(* CODESYS project CtaAppReport_2.0.0.0.library
   Description: Report Library der CTA
   Version: 2.0.0.0
   Title: CtaAppReport
   Author: SIS
   Company: CTA
   Placeholder: CtaAppReport
   DocFormat: reStructuredText
   DefaultNamespace: CtaAppReport
   CompiledLibraryCompatibilityVersion: CODESYS V3.5 SP16 Patch 3
   LanguageModelAttribute: qualified-access-only

Project tree, tasks and I/O mapping:
  libraries: Standard, 3.5.18.0 (System); CtaAppBmk, 2.0.0.0 (CTA); CtaSysConfig, 1.0.0.2 (CTA); CtaVisSymbols, 1.0.0.0 (CTA); CtaSysEvent, 1.0.0.0 (CTA); VisuDialogs, 3.5.16.20 (System); SysFile, 3.5.17.0 (System); SysDir, 3.5.17.0 (System); VisuSymbols, 4.5.0.0 (System); StringUtils, 3.5.18.0 (System); SysTypes2 Interfaces, * (System); TextListUtils, * (System); CtaAppInfluxLog, 1.0.0.1 (CTA); CtaAppTime, 1.0.0.1 (CTA)
  40 Visualizations/
    visualisation REPORT_ID
    TABLE/
      visualisation VIS_REPORT_TABLE
      visualisation VIS_REPORT_TABLE_BASE
      DELETE/
        visualisation VIS_REPORT_DELETE
    PUSHLINE/
      visualisation VIS_REPORT_PUSH_LINE
      visualisation VIS_REPORT_PUSH_LINE_BASE
      visualisation VIS_REPORT_PUSH_LINE_QUERRY
    TABLE LINE/
      visualisation VIS_REPORT_TABLE_LINE_BASE
      visualisation VIS_REPORT_TABLE_LINE_QUERRY
      visualisation VIS_REPORT_TABLE_LINE
    REPORTMANAGER/
      visualisation VIS_REPORTMANAGER
      visualisation VIS_REPORTMANAGER_BASE
    HAND/
      visualisation VIS_REPORT_HAND
    ANZAHL REPORTS/
      visualisation VIS_ANZ_REPORTS_OVERALL
      Modul/
        visualisation VIS_ANZ_REPORTS_MODUL
        visualisation VIS_ANZ_REPORTS_MODUL_BASE
        visualisation VIS_ANZ_REPORTS_MODUL_QUERRY
  30 Program Organization Units/
    CSV/
      function block fbCsvHandler [ST]: metWriteDtFrom, metOpenFile, metCloseFile, FB_INIT, metFillSpace, FB_EXIT, metWriteDtTo, actInitPath, metReadCsv, proGetCountsOfReports, proGetCountOfReportsOnInit, metCreateHeader, proExportIdStart, metExportId, metResetCycleCount, proExport, proIsRegistred, metStartDone, metPrepeareStop, proDenyStop, metCyclicCall, metWriteOnChange, metDeleteHistory, metAddObjForeWriteDtFrom, metAddObjForeWriteDtTo, metAddObjForeWriteOnChange
    OBJ/
      function block fbReportObjectFactory [ST]: metQuittAllReports, metDestroyCsvReportObject, metQuittSelectedReports, metCsvGetItf, metDestroyReportObject, metGetItf, metCreateReportObject, proGetNextPos, proGetAktiveReport, proGetActiveErrorMbString, proIsThereAnAktiveError, proGetActiveWarningMbString, metReSaveAfterDelete, metGarbageControll
      function block fbReportObject [ST]: proGetReporterText, proGetReportText, proAdditionalText, proCountRetry, proIsQuitt, proIsSelected, proMaxRetry, proReportAcknowledgType, proReportId, proReportTextId, proReportTextList, proReportType, proReporterObjectId, proStateActive, proWritePosInCsv, proQuitt, metSendDataToInflux, metReportObject, proReportIn, proDtFrom, proDtTo, proSetMetaData, metDestroy, proPrio, metWriteDtFromToCsv, metWriteDtToToCsv, metSaveOnChange, metGarbage
      function fcWordToHexString [ST]
      function fcReportIdToString8 [ST]
    REPORTER/
      function block fbReportManager [ST]: proWarningText, metSyncReporter, proInfoText, proErrorText, proGetErrorNr, actInit, proGetWarningNr, proGetInfoNr, proAnzError, proAnzWarning, proAnzInfo, proTotalReports
      function block fbReporter [ST]: metGetQuitt, proAktivReport, proHandLokal, proNewReport, metReport, proGetCounts, proDoneReport, proPrio, proOptionalText
    VIS/
      function block fbReportVisu [ST]: metGetReport, metGetShowReport, actConfigFile, proQuittExtern, proMaxOffset, proOffset, actEWI, FB_INIT, metReload, actHistory, actPending, proFilterError, proFilterWarning, proFilterInfo, actCheckFilterAndSort, proAnzReportsInTable, proIdMissmatch
    function fcBmkToId [ST]
    SORT/
      function block fbSort [ST]: metSortPrio, metFilterCustom, proAnzAktiveError, proAnzAktiveInfo, proAnzAktiveReports, proAnzAktiveWarning, proAnzReportsInTable
    program REPORT [ST]
  00000000-0000-0000-0000-000000000000|D:\CoDeSys\LibrariesV3\trunk\Intern\CAA\CAA Template\3.4.0.0 draft\Placeholder.xml
  00000000-0000-0000-0000-000000000000|D:\CoDeSys\LibrariesV3\trunk\Intern\CAA\CAA Template\3.2.0.3 draft\Prefix.pdf
  00000000-0000-0000-0000-000000000000|D:\CoDeSys\LibrariesV3\trunk\Intern\CAA\CAA Template\3.5.2.0 draft\Placeholder.xml
  20 Structs/
    data type enReportType
    data type scPara
    data type scReportMetaData
    data type scReportNr
    data type stReportTextList
    data type enReportacknowledgeType
    data type enTableType
  50 Images/
  10 Documenation/
    global variables VersionHistory
    global variables readMe
  21 Interface/
    interface ITF_REPORTMANAGER: proErrorText, proGetWarningNr, metSyncReporter, proGetErrorNr, proGetInfoNr, proInfoText, proWarningText, proTotalReports
    interface ITF_REPORTOBJECT: proGetReportText, proStateActive, proIsQuitt, proIsSelected, proReportId, proMaxRetry, proCountRetry, proReportTextList, proReportTextId, proReporterObjectId, proAdditionalText, proReportType, proReportAcknowledgType, proWritePosInCsv, proGetReporterText, proReportIn, proDtTo, proDtFrom, metReportObject, proQuitt, proSetMetaData, proPrio, metDestroy, metWriteDtFromToCsv, metSaveOnChange
  11 Library Parameter/
    global variables Parameter
  12 Konstanten/
    global variables GlobalKonstant
  60 Textlisten/
    text list txtLibAp99_1Error
    text list txtLibAp99_2enTypeOfAck
    text list txtLibAp99_2Warnung
    text list txtLibAp99_3Info
    text list GlobalTextList
    text list txtNoTextList
  13 Globale Variablen/
    global variables GVL_Report
    global variables GVL_REPORT_PERSISTENT
*)

// 20 Structs/enReportType
TYPE enReportType :
(
	Info    := 0,
    Warning := 1,
    Error   := 2
);
END_TYPE

// 20 Structs/scPara
TYPE scPara :
    STRUCT
        fbxEnSafetyFernQuitt            :   CtaSysConfig.fbBOOL;
        fbuiMaxFernQuitt                :   CtaSysConfig.fbUINT;         
    END_STRUCT
END_TYPE

// 20 Structs/scReportMetaData
TYPE scReportMetaData :
    STRUCT
        xReportIn                   :   BOOL;                           // Report Input
        xActive                     :   BOOL;                           // State of Report
        xIsQuitt                    :   BOOL;                           // State of Acknowledge
        xQuitt                      :   BOOL;                           // Acknowledge Flag
        xIsSelected                 :   BOOL;                           // State of Selected in Table
        dtFrom                      :   DT;                             // Date and Time of Report happen
        dtTo                        :   DT;                             // Date and Time of Report gone
        iMaxRetry                   :   INT;                            // Max allowed Retries till Acknowledge is required
        iCountRetry                 :   INT;                            // Retries till now
        stReportTxtId               :   STRING[3];                      // Report Id fore Texlist
        stReportTextList            :   STRING[100];                    // Report TextList 
        uliReportId                 :   ULINT;                          // Report Id build out of BMK and Report Text Id. Ex: Bmk 56M111 & Id 3 = 567711103  
        enReportType                :   enReportType;                   // Type of Report
        enReportacknowledgeType     :   enReportacknowledgeType;        // Type of Report Acknowledge
        stReporterObjId             :   STRING[20];                     // Object Id of Reporter      
        stAdditionalText            :   STRING[20];                     // Additional Text
        dwWritePosInCsv             :   DWORD;                          // Position in Csv File fore write dtTo 
        usiPrio                     :   USINT;                          // Prio
    END_STRUCT
END_TYPE

// 20 Structs/scReportNr
TYPE scReportNr :
    STRUCT
        iError              :   INT;            // Error Status
        usiErrorPrio        :   USINT;
        iWarning            :   INT;            // Warning Status
        usiWarnungPrio      :   USINT;
        iInfo               :   INT;            // Info Status
        usiInfoPrio         :   USINT;
    END_STRUCT
END_TYPE

// 20 Structs/stReportTextList
TYPE stReportTextList : STRING[100]; END_TYPE

// 20 Structs/enReportacknowledgeType
TYPE enReportacknowledgeType :
(
	Auto        := 0,
    Quit        := 1,
    RetryN      := 2
);
END_TYPE

// 20 Structs/enTableType
{attribute 'qualified_only'}
{attribute 'strict'}
TYPE enTableType :
(
	PENDING_REPORTS := 0,
    HISTORY_REPORTS := 1
);
END_TYPE

// 10 Documenation/VersionHistory
(* 

.. image:: ../../Images/CTA_Logo.jpg
   :align: right
   :width: 15% 

**Vorlage**   


============ =========== =========== ============================================
**Date**     **Version** **Author**  **Change**
------------ ----------- ----------- --------------------------------------------
04.03.2021   0.0.0.0     SIS         Vorlage erstellt

============ =========== =========== ============================================


*)
VAR_GLOBAL
    stInfo : STRING:= '0.0.0.0, Vorlage, CTA';
END_VAR

// 10 Documenation/readMe
(*

**ReadMe**
 
|	**Empfehlung**
|
|	Die LibAp99aErrorManagement wird benötigt damit aus dem BMK der CTA-E-Schema eine Störungsnummer generiert werden kann. 
|	Es wird für die Ausgabe ein DINT verwendet. Die aufschlüsselung von Buchstaben wird durch die ASCI Nr ersetzt.     
|  
| *Beispiel* 
|
| BMK             =   **56M11**    
| Fehler Nr       =   01-10
| ErrorNr-Modbus  =   BMK    + Fehler Nr
| 56771101        =   567711 + 01
| 56771102        =   567711 + 02
| 56771103        =   567711 + 03
| 56771104        =   567711 + 04
| 56771105        =   567711 + 05
| 56771106        =   567711 + 06
| 56771107        =   567711 + 07 
| 56771108        =   567711 + 08
| 56771109        =   567711 + 09
| 56771110        =   567711 + 10 
|
| Wenn der Fehler keiner BMK zugeordnet werden kann, sollte von der Nr. 1000 hochgezähl werden. 
| Tiefere Nr. werden von den Bibliotheken benötigt. 
*)

VAR_GLOBAL
    xReadMeDone              :   BOOL;
END_VAR

// 13 Globale Variablen/GVL_Report
{attribute 'qualified_only'}
VAR_GLOBAL
    fbReportObjectFactory     :   fbReportObjectFactory;
    fbSort                    :   fbSort;
    fbReportVisu              :   fbReportVisu;
    (* Reports *)             
    ayReportObject            :   ARRAY[1..Parameter.diMaxObject] OF fbReportObject;
    ayItfAktiveReports        :   ARRAY[1..Parameter.diMaxObject] OF ITF_REPORTOBJECT;
    ayItfSortetReportsPrio    :   ARRAY[1..Parameter.diMaxObject] OF ITF_REPORTOBJECT;
    ayItfSortetReportsCustom  :   ARRAY[1..Parameter.diMaxObject] OF ITF_REPORTOBJECT;
    ayCsvReportObject         :   ARRAY[0..GlobalKonstant.iUpperSizeTable] OF fbReportObject;
    fbCsvHandler              :   fbCsvHandler;
    diCountHand               :   DINT;
END_VAR

// 11 Library Parameter/Parameter
{attribute 'qualified_only'}
VAR_GLOBAL CONSTANT
    diMaxObject                  :   DINT :=  50;    // Max 200
    diMaxExportsPerCycle         :   DINT :=  50;    // Kann sich auf die Zykluszeit auswirken wenn zu viele Id pro Zyklus exportiert werden
END_VAR

// 12 Konstanten/GlobalKonstant
{attribute 'qualified_only'}
VAR_GLOBAL CONSTANT
    stTextListWarning           :   stReportTextList    := 'CtaAppReport.txtLibAp99_2Warnung';
    stTextListInfo              :   stReportTextList    := 'CtaAppReport.txtLibAp99_3Info';
    iUpperSizeTable             :   INT                 := 13;   
END_VAR

// 13 Globale Variablen/GVL_REPORT_PERSISTENT
{attribute 'qualified_only'}
VAR_GLOBAL RETAIN 
	scLastErrorReport         :   scReportMetaData;
	scLastWarningReport       :   scReportMetaData;
	scLastInfoReport          :   scReportMetaData;  
END_VAR

// 21 Interface/ITF_REPORTMANAGER
INTERFACE ITF_REPORTMANAGER EXTENDS __SYSTEM.IQueryInterface

PROPERTY proErrorText : STRING[100]
GET
END_GET
END_PROPERTY

PROPERTY proGetWarningNr : INT
GET
END_GET
END_PROPERTY

METHOD metSyncReporter : BOOL
VAR_INPUT
	refFbReporter	:	REFERENCE TO fbReporter;
END_VAR
END_METHOD

PROPERTY proGetErrorNr : INT
GET
END_GET
END_PROPERTY

PROPERTY proGetInfoNr : INT
GET
END_GET
END_PROPERTY

PROPERTY proInfoText : STRING[100]
GET
END_GET
END_PROPERTY

PROPERTY proWarningText : STRING[100]
GET
END_GET
END_PROPERTY

PROPERTY proTotalReports : INT
GET
END_GET
END_PROPERTY

END_INTERFACE

// 30 Program Organization Units/REPORTER/fbReporter
FUNCTION_BLOCK FINAL fbReporter 
VAR
	diArrayReportAdr     :	DINT;
	iCountReports		 :	INT;
	tonDelay			 :	TON;
	tonReset			 :	TON;
	_stReportTextList    :	POINTER TO stReportTextList;
	_iReportID			 :  INT;
	xNewReport			 :  BOOL;
	xAktiveReport		 :  BOOL;
    xDoneReport          :  BOOL;
	_enReportType        :  enReportType;
    xHand                :  BOOL;
    usiPrio              :  USINT;
    xExportDone          :  BOOL; 
    xInitDone            :  BOOL;
END_VAR

METHOD metGetQuitt : BOOL
VAR
    ITF_REPORTOBJECT : ITF_REPORTOBJECT;
END_VAR
IF diArrayReportAdr >= 1 THEN
    IF __QUERYINTERFACE(GVL_Report.fbReportObjectFactory.metGetItf(diArrayReportAdr),ITF_REPORTOBJECT) THEN
        metGetQuitt := ITF_REPORTOBJECT.proIsQuitt;
    END_IF;
ELSE
    metGetQuitt := FALSE;
END_IF
END_METHOD

PROPERTY proAktivReport : BOOL
GET
proAktivReport := xAktiveReport;
END_GET
END_PROPERTY

PROPERTY proHandLokal : BOOL
SET
IF proHandLokal AND  NOT xHand THEN
    GVL_Report.diCountHand := GVL_Report.diCountHand + 1;
    xHand := TRUE;
ELSIF NOT proHandLokal AND xHand THEN
    GVL_Report.diCountHand := GVL_Report.diCountHand - 1;
    IF GVL_Report.diCountHand < 0 THEN
        GVL_Report.diCountHand := 0;
	END_IF;
    xHand := FALSE;    
END_IF;
END_SET
END_PROPERTY

PROPERTY INTERNAL proNewReport : BOOL
SET
xNewReport := proNewReport;
END_SET
GET
proNewReport := xNewReport;
END_GET
END_PROPERTY

METHOD FINAL metReport : BOOL
VAR_INPUT
    xSetReportIn          		:   BOOL;
    iReportID           		:   INT;
    enReportTypeIn      		:   enReportType;
    enReportAcknowledgeTypeIn   :   enReportAcknowledgeType;
	tDelay              		:   TIME;  
	ITF_BMK_IN					:	CtaAppBmk.ITF_BMK;
	pstReportTextListIn 		:	POINTER TO stReportTextList;	 
	stOptionalReportText		:	STRING[20];	
    iRetryTilReportLock 		:   INT;                            
    xResetCount         		:   BOOL;                            
	tReset						:	TIME;                 
END_VAR
VAR
    ITF_REPORTOBJECT            :   ITF_REPORTOBJECT;
END_VAR
IF xInitDone AND_THEN pstReportTextListIn <> 0 AND_THEN ITF_BMK_IN <> 0 THEN
    // Counter mit xResetCount rücksetzen wenn Count < iMaxRetry
    IF tReset > T#0MS AND_THEN enReportAcknowledgeTypeIn = enReportacknowledgeType.RetryN AND_THEN NOT xSetReportIn THEN
        tonReset.IN := iCountReports < iRetryTilReportLock AND iCountReports > 0;
        tonReset.PT	:= tReset;
        tonReset();
	ELSE
		tonReset(IN := FALSE,
				 PT := T#0MS);
    END_IF;
    IF (xResetCount OR tonReset.Q) AND_THEN iCountReports < iRetryTilReportLock AND NOT xSetReportIn  THEN
        diArrayReportAdr := 0;   
        iCountReports := 0;
        tonReset.IN := FALSE;
        tonReset.PT	:= T#0S;	 
        tonReset();
    END_IF;        
	IF xSetReportIn THEN	
		_stReportTextList    := pstReportTextListIn;	
		_iReportID 			 := iReportID;
		_enReportType		 := enReportTypeIn;
	END_IF;
	
	tonDelay.IN          := xSetReportIn;
	tonDelay.PT          := tDelay;
	tonDelay();
	(* Wenn Report nicht registriert Registrierprozess starten *)
    IF diArrayReportAdr = 0 THEN
        // Wenn tonDelay.Q aktiv Registrieren      
        IF tonDelay.Q THEN
            (* Create Report Object *)
            diArrayReportAdr := GVL_Report.fbReportObjectFactory.metCreateReportObject();   
            IF diArrayReportAdr <> 0 THEN 
                IF __QUERYINTERFACE(GVL_Report.fbReportObjectFactory.metGetItf(diArrayReportAdr),ITF_REPORTOBJECT) THEN               
                    (* Set Infos *)  
                    xNewReport := TRUE;
                    xAktiveReport := TRUE;
                    iCountReports := iCountReports + 1;
                    ITF_REPORTOBJECT.proReportType              :=  enReportTypeIn;                         // Report Type
                    ITF_REPORTOBJECT.proReportAcknowledgType    :=  enReportAcknowledgeTypeIn;              // Report Acknowledge Type
                    ITF_REPORTOBJECT.proReportTextId            :=  TO_STRING(iReportID);                   // Report Id
                    ITF_REPORTOBJECT.proReportTextList          :=  pstReportTextListIn^;                   // Report Text list
                    ITF_REPORTOBJECT.proReporterObjectId        :=  ITF_BMK_IN.proGetObjectId;              // Reporter Object Id
                    ITF_REPORTOBJECT.proSetInstancePath         :=  ITF_BMK_IN.proGetInstancePath;          // Reporter Instance Path
                    ITF_REPORTOBJECT.proMaxRetry                :=  iRetryTilReportLock;                    // Max Retries
                    ITF_REPORTOBJECT.proCountRetry              :=  iCountReports;                          // Countet Retries
                    ITF_REPORTOBJECT.proAdditionalText          :=  stOptionalReportText;                   // Additional Text
                    ITF_REPORTOBJECT.proReportIn                :=  xSetReportIn;                           // Report Input
                    ITF_REPORTOBJECT.proPrio                    :=  usiPrio;
                    ITF_REPORTOBJECT.metReportObject();                                                     // Call Object              
                END_IF                                                                 
            END_IF;
        END_IF;
    ELSE
        // Zyklische aktualisierung der Daten nach Registrierung       
        IF __QUERYINTERFACE(GVL_Report.fbReportObjectFactory.metGetItf(diArrayReportAdr),ITF_REPORTOBJECT) THEN
            IF ITF_REPORTOBJECT.proReportIn <> xSetReportIn THEN
                ITF_REPORTOBJECT.proReportIn :=  xSetReportIn;                                   // Report Input
            END_IF;
			// Nach Manuellem Quittieren Counts rücksetzen     
			IF ITF_REPORTOBJECT.proQuitt THEN
				iCountReports := 0;
			END_IF;              
			IF NOT ITF_REPORTOBJECT.proStateActive THEN
                xAktiveReport   := FALSE;   
                xDoneReport     := TRUE;
 
                diArrayReportAdr := 0;  
            END_IF;
            ITF_REPORTOBJECT.metReportObject();                                                             // Call Object 
        ELSE
            diArrayReportAdr := 0;
            xAktiveReport   := FALSE; 
            xDoneReport     := TRUE;
        END_IF;                                              
    END_IF;

    // ID Liste erzeugen
    IF GVL_Report.fbCsvHandler.proExport AND NOT xExportDone THEN
        xExportDone :=  GVL_Report.fbCsvHandler.metExportId(  ITF_BMK_IN	            := 	ITF_BMK_IN,
                                                              iID                       :=  iReportID,
                                                              enReportTypeIn            :=  enReportTypeIn,
                                                              enReportAcknowledgeTypeIn :=  enReportAcknowledgeTypeIn,
                                                              stReportTextListIn        :=  pstReportTextListIn^);
    ELSIF NOT GVL_Report.fbCsvHandler.proExport THEN 
        xExportDone := FALSE;
    END_IF;  
END_IF;
xInitDone := TRUE;
END_METHOD

PROPERTY proGetCounts : INT
GET
proGetCounts := iCountReports;
END_GET
END_PROPERTY

PROPERTY proDoneReport : BOOL
SET
xDoneReport     := proDoneReport;
END_SET
GET
proDoneReport := xDoneReport;
END_GET
END_PROPERTY

PROPERTY proPrio : USINT
SET
IF proPrio <> usiPrio THEN
	usiPrio := proPrio;
END_IF;
END_SET
GET
proPrio := usiPrio;
END_GET
END_PROPERTY

PROPERTY proOptionalText : STRING(20)
GET
VAR
	ITF_REPORTOBJECT : ITF_REPORTOBJECT;
END_VAR
IF diArrayReportAdr <> 0 THEN
	IF __QUERYINTERFACE(GVL_Report.fbReportObjectFactory.metGetItf(diArrayReportAdr),ITF_REPORTOBJECT) THEN 
		proOptionalText := 	ITF_REPORTOBJECT.proAdditionalText;
	END_IF;
END_IF;
END_GET
END_PROPERTY

END_FUNCTION_BLOCK

// 30 Program Organization Units/OBJ/fbReportObjectFactory
FUNCTION_BLOCK fbReportObjectFactory
VAR_INPUT
END_VAR
VAR_OUTPUT
END_VAR
VAR 
    diNextFreePosition            :   DINT := 1;
	dwSync						  :   DWORD;
END_VAR

METHOD metQuittAllReports : BOOL
VAR
    diFor    :   DINT;
END_VAR
FOR diFor := 1 TO Parameter.diMaxObject DO
    IF GVL_Report.ayItfAktiveReports[diFor] <> 0 THEN
        IF GVL_Report.ayItfAktiveReports[diFor].proStateActive AND_THEN NOT GVL_Report.ayItfAktiveReports[diFor].proIsQuitt THEN
            GVL_Report.ayItfAktiveReports[diFor].proQuitt := TRUE;    
		END_IF;
	END_IF;
END_FOR;
END_METHOD

(* Destroy Report Object *)
METHOD PRIVATE metDestroyCsvReportObject : BOOL
VAR_INPUT
    iArrayPos   :   INT;
END_VAR
IF iArrayPos >= 0 AND iArrayPos <= 9 THEN
    GVL_Report.ayCsvReportObject[iArrayPos].metDestroy();
    metDestroyCsvReportObject := TRUE;
END_IF;
END_METHOD

METHOD metQuittSelectedReports : BOOL
VAR
    diFor    :   DINT;
END_VAR
FOR diFor := 1 TO Parameter.diMaxObject DO
    IF GVL_Report.ayItfAktiveReports[diFor] <> 0 THEN
        IF GVL_Report.ayItfAktiveReports[diFor].proIsSelected AND_THEN GVL_Report.ayItfAktiveReports[diFor].proStateActive AND_THEN NOT GVL_Report.ayItfAktiveReports[diFor].proIsQuitt THEN
            GVL_Report.ayItfAktiveReports[diFor].proQuitt := TRUE;    
		END_IF;
	END_IF;
END_FOR;
END_METHOD

METHOD metCsvGetItf : ITF_REPORTOBJECT
VAR_INPUT
    diArrayPos   :   DINT;
END_VAR
IF diArrayPos >= 0 AND diArrayPos <= GlobalKonstant.iUpperSizeTable THEN    
    metCsvGetItf := GVL_Report.ayCsvReportObject[diArrayPos];
END_IF;
END_METHOD

(* Destroy Report Object *)
METHOD PRIVATE metDestroyReportObject : BOOL
VAR_INPUT
    diArrayPos   :   DINT;
END_VAR
IF diArrayPos >= 1 AND diArrayPos <= Parameter.diMaxObject THEN   
    IF NOT GVL_Report.ayReportObject[diArrayPos].proStateActive THEN
        GVL_Report.ayReportObject[diArrayPos].metDestroy();
        metDestroyReportObject := TRUE;
    ELSE
        metDestroyReportObject := FALSE;
    END_IF;
END_IF;
END_METHOD

METHOD metGetItf : ITF_REPORTOBJECT
VAR_INPUT
    diArrayPos   :   DINT;
END_VAR
IF diArrayPos >= 1 AND diArrayPos <= Parameter.diMaxObject THEN
    metGetItf := GVL_Report.ayReportObject[diArrayPos];
END_IF;
END_METHOD

(* Returns Arrayposition of Object*) 
METHOD metCreateReportObject : DINT
VAR
    diCurrentPositon    :   DINT;
    diCurrentOverFlows  :   DINT;
    diSavetyCount       :   DINT;
	dwExklusiveAcces	:	DWORD;
END_VAR
REPEAT 
    metCreateReportObject := 0;
	dwExklusiveAcces := TEST_AND_SET(dwSync);
	IF dwExklusiveAcces = 0 THEN
		IF diNextFreePosition + 1 > Parameter.diMaxObject THEN
			diCurrentPositon    := __XADD(ADR(diNextFreePosition),-Parameter.diMaxObject + 1);
		ELSE
			diCurrentPositon := __XADD(ADR(diNextFreePosition),1);  
		END_IF;
		dwSync := 0;
	END_IF;
    IF diCurrentPositon >= 1 AND diCurrentPositon <= Parameter.diMaxObject THEN
        IF NOT GVL_Report.ayReportObject[diCurrentPositon].proStateActive THEN
            metDestroyReportObject(diCurrentPositon);
            metCreateReportObject := diCurrentPositon;     
            metDestroyReportObject(diNextFreePosition);
        END_IF;
    END_IF;
    diSavetyCount := diSavetyCount + 1;
UNTIL
    metCreateReportObject <> 0 OR diSavetyCount >= Parameter.diMaxObject
END_REPEAT;
END_METHOD

PROPERTY proGetNextPos : DINT
GET
proGetNextPos := diNextFreePosition;
END_GET
END_PROPERTY

PROPERTY proGetAktiveReport : ITF_REPORTOBJECT
GET
proGetAktiveReport := GVL_Report.ayItfSortetReportsPrio[1];
END_GET
END_PROPERTY

PROPERTY proGetActiveErrorMbString : STRING(160)
GET
VAR
    ITF_REPORTOBJECT_TEMP   :   ITF_REPORTOBJECT;
END_VAR
(* Error Nr as String *)
proGetActiveErrorMbString := '';
IF __QUERYINTERFACE(proGetAktiveReport,ITF_REPORTOBJECT_TEMP) THEN
    IF ITF_REPORTOBJECT_TEMP.proReportType = enReportType.Error THEN
        proGetActiveErrorMbString := CONCAT(fcReportIdToString8(ITF_REPORTOBJECT_TEMP.proReportId),CONCAT(' ',CONCAT(ITF_REPORTOBJECT_TEMP.proGetBMK,CONCAT(' ',ITF_REPORTOBJECT_TEMP.proGetReportText))));       
    ELSE
        RETURN;
	END_IF;
END_IF;
END_GET
END_PROPERTY

PROPERTY proIsThereAnAktiveError : BOOL
GET
VAR
    diFor   :   DINT;
END_VAR
proIsThereAnAktiveError := FALSE;
FOR diFor := 1 TO Parameter.diMaxObject DO
    IF GVL_Report.ayItfSortetReportsPrio[diFor] <> 0 THEN
        IF GVL_Report.ayItfSortetReportsPrio[diFor].proStateActive THEN
            IF GVL_Report.ayItfSortetReportsPrio[diFor].proReportType = enReportType.Error THEN
                proIsThereAnAktiveError := TRUE;
                EXIT;    
            ELSE
                CONTINUE;
            END_IF;
        ELSE
            CONTINUE;
        END_IF;
    ELSE
        CONTINUE;
    END_IF;
END_FOR;
END_GET
END_PROPERTY

PROPERTY proGetActiveWarningMbString : STRING(160)
GET
VAR
    ITF_REPORTOBJECT_TEMP   :   ITF_REPORTOBJECT;
    diFor                   :   DINT;
END_VAR
(* Error Nr as String *)
proGetActiveWarningMbString := '';
// Warning
FOR diFor := Parameter.diMaxObject TO 1 BY -1 DO 
    IF GVL_Report.ayItfSortetReportsPrio[diFor] <> 0 AND_THEN GVL_Report.ayItfSortetReportsPrio[diFor].proStateActive AND_THEN GVL_Report.ayItfSortetReportsPrio[diFor].proReportType = enReportType.Warning THEN
        ITF_REPORTOBJECT_TEMP :=  GVL_Report.ayItfSortetReportsPrio[diFor];   
        RETURN;
    END_IF;        
END_FOR;
IF ITF_REPORTOBJECT_TEMP <> 0 THEN
        proGetActiveWarningMbString := CONCAT(fcReportIdToString8(ITF_REPORTOBJECT_TEMP.proReportId),CONCAT(' ',CONCAT(ITF_REPORTOBJECT_TEMP.proGetBMK,CONCAT(' ',ITF_REPORTOBJECT_TEMP.proGetReportText))));       
END_IF;
END_GET
END_PROPERTY

METHOD metReSaveAfterDelete : BOOL
VAR
    diFor    :   DINT;
END_VAR
FOR diFor := 1 TO Parameter.diMaxObject DO
    IF GVL_Report.ayItfAktiveReports[diFor] <> 0 THEN
        GVL_Report.ayItfAktiveReports[diFor].metWriteDtFromToCsv(); 
	END_IF;
END_FOR;
END_METHOD

METHOD metGarbageControll : BOOL
VAR
    diFor   :   DINT;
END_VAR
metGarbageControll := FALSE;   
FOR diFor := 1 TO Parameter.diMaxObject DO
    IF GVL_Report.ayReportObject[diFor].proStateActive THEN
        IF GVL_Report.ayReportObject[diFor].metGarbage() THEN     
        	metGarbageControll := TRUE;   
		END_IF;
	END_IF;
END_FOR;
END_METHOD

END_FUNCTION_BLOCK

// 30 Program Organization Units/REPORT
PROGRAM REPORT
VAR
END_VAR

(* Csv Fb *)
GVL_Report.fbCsvHandler();
(* Visu Fb *)
GVL_Report.fbReportVisu();
(* Prüfen ob Objecte Unbrauchbar sind *)
IF GVL_Report.fbReportObjectFactory.metGarbageControll() THEN
	(* Tabelle neu Laden wenn Objecte zerstört *)
    GVL_Report.fbSort.metSortPrio();
END_IF;

END_PROGRAM

// 30 Program Organization Units/CSV/fbCsvHandler
FUNCTION_BLOCK fbCsvHandler IMPLEMENTS CtaSysEvent.ITF_APPEVENT
VAR CONSTANT
    wSize               :   WORD    :=  786;  
    wSizeHeader         :   WORD    :=  150;
END_VAR
VAR
	stFilePathHistory   :   STRING;
    stFileDownloadHtml  :   STRING;
    stFilePathDelete    :   STRING;
    xInitDone           :   BOOL;
    xIsNotSimulation    :   BOOL;
    stSpace             :   STRING[1] := ' ';
    stRN                :   STRING[1] := '$R';
    stSC                :   STRING[1] := ';';
    stHeader            :   STRING[wSizeHeader]; 
    stHtmlDownload      :   STRING[88];
    RTS_IEC_RESULT_Ini  :   RTS_IEC_RESULT;
    RTS_IEC_HANDLE_Ini  :   RTS_IEC_HANDLE;     
    RTS_IEC_RESULT_Csv  :   RTS_IEC_RESULT;
    RTS_IEC_HANDLE_Csv  :   RTS_IEC_HANDLE;     
    RTS_IEC_RESULT_Exp  :   RTS_IEC_RESULT;
    RTS_IEC_HANDLE_ExE  :   RTS_IEC_HANDLE; 
    RTS_IEC_HANDLE_ExW  :   RTS_IEC_HANDLE;    
    RTS_IEC_HANDLE_ExI  :   RTS_IEC_HANDLE;   
    FILE_STATUS         :   SysFile.SYS_FILE_STATUS; 
    xExportId           :   BOOL;
    xExportPossible     :   BOOL;
    xIsExporting        :   BOOL;
    xExportDoneTemp     :   BOOL;
    xExportDone         :   BOOL;
    udiSizeOfFileOnInit :   UDINT;
    udiSizeOfFileNow    :   UDINT;
    dwWrite             :   DWORD;
    diCountExp          :   DINT;
    iWait               :   INT;
    xIsRegistretAppEvent:   BOOL;
    ITF_BMK_NEXT_EXPORT :   CtaAppBmk.ITF_BMK;
	udiOldValueCounts	:	UDINT;
	dwSync				:	DWORD;
	ayITF_WriteDtFrom	:	ARRAY[0..Parameter.diMaxObject] OF ITF_REPORTOBJECT;
	diNextFreeDtFrom	:	DINT;
	diNextFreeDtFromOld	:	DINT;
	ayITF_WriteDtTo		:	ARRAY[0..Parameter.diMaxObject] OF ITF_REPORTOBJECT;
	diNextFreeDtTo		:	DINT;
	diNextFreeDtToOld	:	DINT;
	ayITF_WriteChange	:	ARRAY[0..Parameter.diMaxObject] OF ITF_REPORTOBJECT;
	diNextFreeChange	:	DINT;
	diNextFreeChangeOld	:	DINT;
	diFor				:	DINT;

END_VAR;

(* Dt From *)
IF diNextFreeDtFrom <> diNextFreeDtFromOld THEN
	FOR diFor := LOWER_BOUND(ayITF_WriteDtFrom,1) TO UPPER_BOUND(ayITF_WriteDtFrom,1) DO
		IF ayITF_WriteDtFrom[diFor] <> 0 THEN
			metWriteDtFrom(ayITF_WriteDtFrom[diFor]);
			ayITF_WriteDtFrom[diFor] := 0;
		END_IF;
	END_FOR;
	diNextFreeDtFromOld := diNextFreeDtFrom;
ELSE
	diNextFreeDtFrom 	:= 0;
	diNextFreeDtFromOld	:= 0;
END_IF;

(* Change *)
IF diNextFreeChange <> diNextFreeChangeOld THEN
	FOR diFor := LOWER_BOUND(ayITF_WriteChange,1) TO UPPER_BOUND(ayITF_WriteChange,1) DO
		IF ayITF_WriteChange[diFor] <> 0 THEN
			metWriteOnChange(ayITF_WriteChange[diFor],ayITF_WriteChange[diFor].proWritePosInCsv);
			ayITF_WriteChange[diFor] := 0;
		END_IF;
	END_FOR;
	diNextFreeChangeOld := diNextFreeChange;
ELSE
	diNextFreeChange 	:= 0;
	diNextFreeChangeOld	:= 0;	
END_IF;

(* DtTo *)
IF diNextFreeDtTo <> diNextFreeDtToOld THEN
	FOR diFor := LOWER_BOUND(ayITF_WriteDtTo,1) TO UPPER_BOUND(ayITF_WriteDtTo,1)  DO
		IF ayITF_WriteDtTo[diFor] <> 0 THEN
			metWriteDtTo(ayITF_WriteDtTo[diFor],ayITF_WriteDtTo[diFor].proWritePosInCsv);
			ayITF_WriteDtTo[diFor] := 0;
		END_IF;
	END_FOR;
	diNextFreeDtToOld := diNextFreeDtTo;
ELSE
	diNextFreeDtTo 		:= 0;
	diNextFreeDtToOld	:= 0;	
END_IF;

METHOD PRIVATE metWriteDtFrom : DWORD
VAR_INPUT
    ITF_REPORTOBJECT_IN : ITF_REPORTOBJECT;
END_VAR
VAR
    ITF_REPORTOBJECT_QUERY  :   ITF_REPORTOBJECT;
    stTemp          :   STRING[255];
    dwIstPso        :   DWORD;    
	pstDataToWriteF :   POINTER TO STRING[wSize];
	diFor           :   DINT;
END_VAR
IF __QUERYINTERFACE(ITF_REPORTOBJECT_IN,ITF_REPORTOBJECT_QUERY) AND wSize <> 0 THEN
    pstDataToWriteF := __NEW(STRING[wSize]);
    IF pstDataToWriteF <> 0 THEN  
        // Daten zum Schreiben erzeugen  
        pstDataToWriteF^  :=    '';
        stTemp := '';
        IF ITF_REPORTOBJECT_QUERY.proReportType = enReportType.Error THEN
            stTemp := 'ERROR';
        ELSIF ITF_REPORTOBJECT_QUERY.proReportType = enReportType.Warning THEN
            stTemp := 'WARNING';
        ELSIF ITF_REPORTOBJECT_QUERY.proReportType = enReportType.Info THEN
            stTemp := 'INFO';
        END_IF;
        metFillSpace(stTemp,7);
        StrConcatA(ADR(stTemp),pstDataToWriteF,TO_INT(SIZEOF(pstDataToWriteF^)));  
        stTemp := '';
        stTemp := stSC;
        StrConcatA(ADR(stTemp),pstDataToWriteF,TO_INT(SIZEOF(pstDataToWriteF^)));     
        stTemp := '';
        stTemp := TO_STRING(ITF_REPORTOBJECT_QUERY.proReportId);
        metFillSpace(stTemp,10);
        StrConcatA(ADR(stTemp),pstDataToWriteF,TO_INT(SIZEOF(pstDataToWriteF^)));    
        stTemp := '';
        stTemp := stSC;
        StrConcatA(ADR(stTemp),pstDataToWriteF,TO_INT(SIZEOF(pstDataToWriteF^)));                    
        stTemp := '';
        stTemp := TO_STRING(ITF_REPORTOBJECT_QUERY.proGetReporterText);
        metFillSpace(stTemp,150);
        StrConcatA(ADR(stTemp),pstDataToWriteF,TO_INT(SIZEOF(pstDataToWriteF^)));                                        
        stTemp := '';
        stTemp := stSC;
        StrConcatA(ADR(stTemp),pstDataToWriteF,TO_INT(SIZEOF(pstDataToWriteF^)));
        stTemp := '';
        stTemp := TO_STRING(ITF_REPORTOBJECT_QUERY.proGetReportText);
        metFillSpace(stTemp,140); 
        StrConcatA(ADR(stTemp),pstDataToWriteF,TO_INT(SIZEOF(pstDataToWriteF^)));               
        stTemp := '';
        stTemp := stSC;
        StrConcatA(ADR(stTemp),pstDataToWriteF,TO_INT(SIZEOF(pstDataToWriteF^)));        
        stTemp := '';
        stTemp := TO_STRING(ITF_REPORTOBJECT_QUERY.proDtFrom);
        metFillSpace(stTemp,22);
        StrConcatA(ADR(stTemp),pstDataToWriteF,TO_INT(SIZEOF(pstDataToWriteF^)));  
        stTemp := '';
        stTemp := stSC;
        StrConcatA(ADR(stTemp),pstDataToWriteF,TO_INT(SIZEOF(pstDataToWriteF^)));
        stTemp := '';           // Dt To = lehr
        metFillSpace(stTemp,22);
        StrConcatA(ADR(stTemp),pstDataToWriteF,TO_INT(SIZEOF(pstDataToWriteF^))); 
        stTemp := '';
        stTemp := stSC;
        StrConcatA(ADR(stTemp),pstDataToWriteF,TO_INT(SIZEOF(pstDataToWriteF^)));
        stTemp := '';
        stTemp := TO_STRING(ITF_REPORTOBJECT_QUERY.proIsQuitt);
        metFillSpace(stTemp,5);
        StrConcatA(ADR(stTemp),pstDataToWriteF,TO_INT(SIZEOF(pstDataToWriteF^))); 
        stTemp := '';
        stTemp := stSC;
        StrConcatA(ADR(stTemp),pstDataToWriteF,TO_INT(SIZEOF(pstDataToWriteF^)));
        stTemp := '';
        stTemp := TO_STRING(ITF_REPORTOBJECT_QUERY.proReportTextList);
        metFillSpace(stTemp,100);
        StrConcatA(ADR(stTemp),pstDataToWriteF,TO_INT(SIZEOF(pstDataToWriteF^))); 
        stTemp := '';
        stTemp := stSC;
        StrConcatA(ADR(stTemp),pstDataToWriteF,TO_INT(SIZEOF(pstDataToWriteF^)));
        stTemp := '';
        stTemp := TO_STRING(ITF_REPORTOBJECT_QUERY.proReportTextId);
        metFillSpace(stTemp,3);
        StrConcatA(ADR(stTemp),pstDataToWriteF,TO_INT(SIZEOF(pstDataToWriteF^)));                       
        stTemp := '';
        stTemp := stSC;
        StrConcatA(ADR(stTemp),pstDataToWriteF,TO_INT(SIZEOF(pstDataToWriteF^)));
        stTemp := '';
        stTemp := TO_STRING(TO_USINT(ITF_REPORTOBJECT_QUERY.proReportAcknowledgType));
        metFillSpace(stTemp,3);
        StrConcatA(ADR(stTemp),pstDataToWriteF,TO_INT(SIZEOF(pstDataToWriteF^)));
        stTemp := '';
        stTemp := stSC;
        StrConcatA(ADR(stTemp),pstDataToWriteF,TO_INT(SIZEOF(pstDataToWriteF^)));
        stTemp := '';
        stTemp := ITF_REPORTOBJECT_QUERY.proGetObjectId;
        metFillSpace(stTemp,20);        
        StrConcatA(ADR(stTemp),pstDataToWriteF,TO_INT(SIZEOF(pstDataToWriteF^))); 
        stTemp := '';
        stTemp := stSC;
        StrConcatA(ADR(stTemp),pstDataToWriteF,TO_INT(SIZEOF(pstDataToWriteF^)));
        stTemp := '';
        stTemp := ITF_REPORTOBJECT_QUERY.proGetInstancePath;
        metFillSpace(stTemp,255);      
        StrConcatA(ADR(stTemp),pstDataToWriteF,TO_INT(SIZEOF(pstDataToWriteF^)));
        stTemp := '';
        stTemp := stSC;
        StrConcatA(ADR(stTemp),pstDataToWriteF,TO_INT(SIZEOF(pstDataToWriteF^)));
        stTemp := '';
        stTemp := ITF_REPORTOBJECT_QUERY.proAdditionalText;
        metFillSpace(stTemp,20);
        StrConcatA(ADR(stTemp),pstDataToWriteF,TO_INT(SIZEOF(pstDataToWriteF^)));
        stTemp := '';
        stTemp := stSC;
        StrConcatA(ADR(stTemp),pstDataToWriteF,TO_INT(SIZEOF(pstDataToWriteF^)));        
        stTemp := '';
        stTemp := TO_STRING(ITF_REPORTOBJECT_QUERY.proPrio);
        metFillSpace(stTemp,3); 
        StrConcatA(ADR(stTemp),pstDataToWriteF,TO_INT(SIZEOF(pstDataToWriteF^)));   
        stTemp := '';
        stTemp := stSC;
        StrConcatA(ADR(stTemp),pstDataToWriteF,TO_INT(SIZEOF(pstDataToWriteF^)));
        stTemp := '';
        stTemp := TO_STRING(ITF_REPORTOBJECT_QUERY.proReportIn);
        metFillSpace(stTemp,5);    
        StrConcatA(ADR(stTemp),pstDataToWriteF,TO_INT(SIZEOF(pstDataToWriteF^)));       
        stTemp := '';
        stTemp := stSC;
        StrConcatA(ADR(stTemp),pstDataToWriteF,TO_INT(SIZEOF(pstDataToWriteF^)));
        stTemp := '';
        stTemp := TO_STRING(ITF_REPORTOBJECT_QUERY.proStateActive);
        metFillSpace(stTemp,5);    
        StrConcatA(ADR(stTemp),pstDataToWriteF,TO_INT(SIZEOF(pstDataToWriteF^)));       
        (* String mit Lehrzeichen auffüllen und mit $R abschliessen *)                     
        FOR diFor := StrLenA(pstDataToWriteF) TO wSize -1 DO
            IF diFor < wSize -1 THEN
                pstDataToWriteF^[diFor] := stSpace[0];
            ELSE
                pstDataToWriteF^[diFor] := stRN[0];
            END_IF;
        END_FOR;                          
        // Daten Schreiben
        dwWrite := 0;
        IF metOpenFile() THEN   
            // Grösse Ermitteln
            metWriteDtFrom    := TO_DWORD(SysFile.SysFileGetSizeByHandle(RTS_IEC_HANDLE_Csv,ADR(RTS_IEC_RESULT_Csv)));        
            SysFile.SysFileSetPos(RTS_IEC_HANDLE_CSv,metWriteDtFrom);
            SysFile.SysFileGetPos(RTS_IEC_HANDLE_Csv,ADR(dwIstPso)); 
            IF metWriteDtFrom = dwIstPso THEN  
                dwWrite := TO_DWORD(SysFile.SysFileWrite(RTS_IEC_HANDLE_Csv,pstDataToWriteF,SIZEOF(pstDataToWriteF^)-1,ADR(RTS_IEC_RESULT_Csv)));
            END_IF;
			ITF_REPORTOBJECT_IN.proWritePosInCsv := metWriteDtFrom;
        END_IF;     
        __DELETE(pstDataToWriteF);
    END_IF;
END_IF;
END_METHOD

METHOD PRIVATE metOpenFile : BOOL
VAR_INPUT
END_VAR
IF RTS_IEC_HANDLE_Csv = 0 THEN
	__TRY
		RTS_IEC_HANDLE_Csv := SysFile.SysFileOpen(stFilePathHistory,SysFile.ACCESS_MODE.AM_READ_PLUS,ADR(RTS_IEC_RESULT_Csv)); 
		FILE_STATUS := SysFile.SysFileGetStatus2(RTS_IEC_HANDLE_Csv,ADR(RTS_IEC_RESULT_Csv));
	__CATCH
		RTS_IEC_HANDLE_Csv := 0;
	__ENDTRY
END_IF;

IF RTS_IEC_HANDLE_Csv <> 0 AND RTS_IEC_RESULT_Csv = 0 AND FILE_STATUS = SysFile.SYS_FILE_STATUS.FS_OK THEN
    metOpenFile := TRUE;
ELSE
    metOpenFile := FALSE;
    RTS_IEC_HANDLE_Csv := 0;
END_IF;
END_METHOD

METHOD PRIVATE metCloseFile : BOOL
VAR_INPUT
END_VAR
IF RTS_IEC_HANDLE_Csv <> 0 THEN
	__TRY
    	SysFile.SysFileClose(RTS_IEC_HANDLE_Csv);
	__CATCH
		RTS_IEC_HANDLE_Csv := 0;  	
	__ENDTRY
    RTS_IEC_HANDLE_Csv := 0;    
END_IF;
END_METHOD

//FB_Init ist immer implizit verfügbar und wird primär für die Initialisierung verwendet.
//Der Rückgabewert wird nicht ausgewertet. Für gezielte Einflussnahme können Sie
//die Methoden explizit deklarieren und darin mit dem Standard-Initialisierungscode 
//zusätzlichen Code bereitstellen. Sie können den Rückgabewert auswerten.
METHOD FB_Init: BOOL
VAR_INPUT    
bInitRetains: BOOL; // TRUE: Die Retain-Variablen werden initialisiert (Reset warm / Reset kalt)    
bInCopyCode: BOOL;  // TRUE: Die Instanz wird danach in den Kopiercode kopiert (Online-Change)
END_VAR
actInitPath();
CtaSysEvent.fcRegistry(THIS^);
END_METHOD

METHOD PRIVATE metFillSpace : BOOL
VAR_INPUT
    stIn        :   REFERENCE TO STRING[255];
    iSize       :   INT;
END_VAR
VAR
    iFor        :   INT;
END_VAR
FOR iFor := LEN(stIn) TO iSize -1 DO
    stIn[iFor]      := 32;
    stIn[iFor+1]    := 0;
END_FOR;
END_METHOD

//FB_Exit muss explizit implementiert werden. Wenn es eine Implementierung gibt, dann wird 
//die Methode aufgerufen, bevor die Steuerung den Code der Funktionsbaustein-Instanz entfernt
//(impliziter Aufruf. Der Rückgabewert wird nicht ausgewertet.
METHOD FB_Exit: BOOL
VAR_INPUT    
bInCopyCode: BOOL;  // TRUE: Die Exit-Methode wird aufgerufen, um die Instanz zu verlassen, die hinterher kopiert wird Online-Change).  
END_VAR
IF NOT bInCopyCode THEN
    metCloseFile();
END_IF;
END_METHOD

METHOD PRIVATE metWriteDtTo : BOOL
VAR_INPUT
    ITF_REPORTOBJECT_IN : ITF_REPORTOBJECT;
    dwWritePos   :   DWORD;
END_VAR
VAR
    ITF_REPORTOBJECT_QUERY  :   ITF_REPORTOBJECT;
    stTemp          :   STRING[255];
    dwIstPso        :   DWORD;
	pstDataToWriteT     :   POINTER TO STRING[wSize]; 
	diFor               :   DINT;	

END_VAR
IF __QUERYINTERFACE(ITF_REPORTOBJECT_IN,ITF_REPORTOBJECT_QUERY) AND wSize <> 0  THEN
    pstDataToWriteT := __NEW(STRING[wSize]);
    IF pstDataToWriteT <> 0 THEN    
        // Daten zum Schreiben erzeugen
        pstDataToWriteT^  :=    '';
        stTemp := '';
        IF ITF_REPORTOBJECT_QUERY.proReportType = enReportType.Error THEN
            stTemp := 'ERROR';
        ELSIF ITF_REPORTOBJECT_QUERY.proReportType = enReportType.Warning THEN
            stTemp := 'WARNING';
        ELSIF ITF_REPORTOBJECT_QUERY.proReportType = enReportType.Info THEN
            stTemp := 'INFO';
        END_IF;
        metFillSpace(stTemp,7);
        StrConcatA(ADR(stTemp),pstDataToWriteT,TO_INT(SIZEOF(pstDataToWriteT^)));  
        stTemp := '';
        stTemp := stSC;
        StrConcatA(ADR(stTemp),pstDataToWriteT,TO_INT(SIZEOF(pstDataToWriteT^)));     
        stTemp := '';
        stTemp := TO_STRING(ITF_REPORTOBJECT_QUERY.proReportId);
        metFillSpace(stTemp,10);
        StrConcatA(ADR(stTemp),pstDataToWriteT,TO_INT(SIZEOF(pstDataToWriteT^)));    
        stTemp := '';
        stTemp := stSC;
        StrConcatA(ADR(stTemp),pstDataToWriteT,TO_INT(SIZEOF(pstDataToWriteT^)));                    
        stTemp := '';
        stTemp := TO_STRING(ITF_REPORTOBJECT_QUERY.proGetReporterText);
        metFillSpace(stTemp,150);
        StrConcatA(ADR(stTemp),pstDataToWriteT,TO_INT(SIZEOF(pstDataToWriteT^)));                                        
        stTemp := '';
        stTemp := stSC;
        StrConcatA(ADR(stTemp),pstDataToWriteT,TO_INT(SIZEOF(pstDataToWriteT^)));
        stTemp := '';
        stTemp := TO_STRING(ITF_REPORTOBJECT_QUERY.proGetReportText);
        metFillSpace(stTemp,140); 
        StrConcatA(ADR(stTemp),pstDataToWriteT,TO_INT(SIZEOF(pstDataToWriteT^)));               
        stTemp := '';
        stTemp := stSC;
        StrConcatA(ADR(stTemp),pstDataToWriteT,TO_INT(SIZEOF(pstDataToWriteT^)));        
        stTemp := '';
        stTemp := TO_STRING(ITF_REPORTOBJECT_QUERY.proDtFrom);
        metFillSpace(stTemp,22);
        StrConcatA(ADR(stTemp),pstDataToWriteT,TO_INT(SIZEOF(pstDataToWriteT^)));  
        stTemp := '';
        stTemp := stSC;
        StrConcatA(ADR(stTemp),pstDataToWriteT,TO_INT(SIZEOF(pstDataToWriteT^)));
        stTemp := TO_STRING(ITF_REPORTOBJECT_QUERY.proDtTo);
        metFillSpace(stTemp,22);
        StrConcatA(ADR(stTemp),pstDataToWriteT,TO_INT(SIZEOF(pstDataToWriteT^))); 
        stTemp := '';
        stTemp := stSC;
        StrConcatA(ADR(stTemp),pstDataToWriteT,TO_INT(SIZEOF(pstDataToWriteT^)));
        stTemp := '';
        stTemp := TO_STRING(ITF_REPORTOBJECT_QUERY.proIsQuitt);
        metFillSpace(stTemp,5);
        StrConcatA(ADR(stTemp),pstDataToWriteT,TO_INT(SIZEOF(pstDataToWriteT^))); 
        stTemp := '';
        stTemp := stSC;
        StrConcatA(ADR(stTemp),pstDataToWriteT,TO_INT(SIZEOF(pstDataToWriteT^)));
        stTemp := '';
        stTemp := TO_STRING(ITF_REPORTOBJECT_QUERY.proReportTextList);
        metFillSpace(stTemp,100);
        StrConcatA(ADR(stTemp),pstDataToWriteT,TO_INT(SIZEOF(pstDataToWriteT^))); 
        stTemp := '';
        stTemp := stSC;
        StrConcatA(ADR(stTemp),pstDataToWriteT,TO_INT(SIZEOF(pstDataToWriteT^)));
        stTemp := '';
        stTemp := TO_STRING(ITF_REPORTOBJECT_QUERY.proReportTextId);
        metFillSpace(stTemp,3);
        StrConcatA(ADR(stTemp),pstDataToWriteT,TO_INT(SIZEOF(pstDataToWriteT^)));                       
        stTemp := '';
        stTemp := stSC;
        StrConcatA(ADR(stTemp),pstDataToWriteT,TO_INT(SIZEOF(pstDataToWriteT^)));
        stTemp := '';
        stTemp := TO_STRING(TO_USINT(ITF_REPORTOBJECT_QUERY.proReportAcknowledgType));
        metFillSpace(stTemp,3);
        StrConcatA(ADR(stTemp),pstDataToWriteT,TO_INT(SIZEOF(pstDataToWriteT^)));
        stTemp := '';
        stTemp := stSC;
        StrConcatA(ADR(stTemp),pstDataToWriteT,TO_INT(SIZEOF(pstDataToWriteT^)));
        stTemp := '';
        stTemp := ITF_REPORTOBJECT_QUERY.proGetObjectId;
        metFillSpace(stTemp,20);        
        StrConcatA(ADR(stTemp),pstDataToWriteT,TO_INT(SIZEOF(pstDataToWriteT^))); 
        stTemp := '';
        stTemp := stSC;
        StrConcatA(ADR(stTemp),pstDataToWriteT,TO_INT(SIZEOF(pstDataToWriteT^)));
        stTemp := '';
        stTemp := ITF_REPORTOBJECT_QUERY.proGetInstancePath;
        metFillSpace(stTemp,255);      
        StrConcatA(ADR(stTemp),pstDataToWriteT,TO_INT(SIZEOF(pstDataToWriteT^)));
        stTemp := '';
        stTemp := stSC;
        StrConcatA(ADR(stTemp),pstDataToWriteT,TO_INT(SIZEOF(pstDataToWriteT^)));
        stTemp := '';
        stTemp := ITF_REPORTOBJECT_QUERY.proAdditionalText;
        metFillSpace(stTemp,20);
        StrConcatA(ADR(stTemp),pstDataToWriteT,TO_INT(SIZEOF(pstDataToWriteT^)));
        stTemp := '';
        stTemp := stSC;
        StrConcatA(ADR(stTemp),pstDataToWriteT,TO_INT(SIZEOF(pstDataToWriteT^)));            
        stTemp := '';
        stTemp := TO_STRING(ITF_REPORTOBJECT_QUERY.proPrio);
        metFillSpace(stTemp,3); 
        StrConcatA(ADR(stTemp),pstDataToWriteT,TO_INT(SIZEOF(pstDataToWriteT^)));      
        stTemp := '';
        stTemp := stSC;
        StrConcatA(ADR(stTemp),pstDataToWriteT,TO_INT(SIZEOF(pstDataToWriteT^)));
        stTemp := '';
        stTemp := TO_STRING(ITF_REPORTOBJECT_QUERY.proReportIn);
        metFillSpace(stTemp,5);                
        StrConcatA(ADR(stTemp),pstDataToWriteT,TO_INT(SIZEOF(pstDataToWriteT^))); 
        stTemp := '';
        stTemp := stSC;
        StrConcatA(ADR(stTemp),pstDataToWriteT,TO_INT(SIZEOF(pstDataToWriteT^)));
        stTemp := '';
        stTemp := TO_STRING(ITF_REPORTOBJECT_QUERY.proStateActive);
        metFillSpace(stTemp,5);                
        StrConcatA(ADR(stTemp),pstDataToWriteT,TO_INT(SIZEOF(pstDataToWriteT^)));         
        (* String mit Lehrzeichen auffüllen und mit $R abschliessen *)                     
        FOR diFor := StrLenA(pstDataToWriteT) TO wSize -1 DO
            IF diFor < wSize -1 THEN
                pstDataToWriteT^[diFor] := stSpace[0];
            ELSE
                pstDataToWriteT^[diFor] := stRN[0];
            END_IF;
        END_FOR;                          
        // Daten Schreiben
        IF metOpenFile() THEN
            SysFile.SysFileSetPos(RTS_IEC_HANDLE_Csv,dwWritePos);
            SysFile.SysFileGetPos(RTS_IEC_HANDLE_Csv,ADR(dwIstPso));       
			IF dwWritePos = dwIstPso THEN   
            	dwWrite := TO_DWORD(SysFile.SysFileWrite(RTS_IEC_HANDLE_Csv,pstDataToWriteT,SIZEOF(pstDataToWriteT^)-1,ADR(RTS_IEC_RESULT_Csv)));
			END_IF;	
        END_IF;
        __DELETE(pstDataToWriteT);
    END_IF;
END_IF;
END_METHOD

ACTION actInitPath:
IF NOT xInitDone THEN
	__TRY
    {IF NOT defined (IsSimulationMode)}
        // FILE Path auf SPS
        stFilePathHistory  :=       CONCAT(
                                    CONCAT(
                                            './visu/History/Export/',
                                            'EWI_History'),
                                            '.csv');   
        stFileDownloadHtml  :=  './visu/History/HistoryDownload.htm';                                    
        xIsNotSimulation := TRUE;    
    {ELSE}
        // FILE Path auf Laptop
        stFilePathHistory  :=       CONCAT(
                                    CONCAT(
                                    CONCAT(                            
                                            'C:/PFC_Simulation/visu/',
                                            'History/Export/'),
                                            'EWI_History'),
                                            '.csv');                                                        
    {END_IF}   
    // Download Html erzeugen
    IF xIsNotSimulation THEN
        (* History Download *)
            RTS_IEC_HANDLE_Ini := SysFile.SysFileOpen(stFileDownloadHtml,SysFile.ACCESS_MODE.AM_WRITE_PLUS,ADR(RTS_IEC_RESULT_Ini));   
            // Schreibe Position festlegen
            SysFile.SysFileSetPos(RTS_IEC_HANDLE_Ini,0);  
            stHtmlDownload  := '';      
            stHtmlDownload  := '<HTML><HEAD><TITLE></TITLE></HEAD><BODY>';
            // Daten Schreiben
            SysFile.SysFileWrite(RTS_IEC_HANDLE_Ini,ADR(stHtmlDownload),TO_DWORD(LEN(stHtmlDownload)),ADR(RTS_IEC_RESULT_Ini));  
            stHtmlDownload  := '';      
            stHtmlDownload  := '<a href="Export/EWI_History.csv" download = "EWI_History.csv">History Download</a><br />';    
            // Daten Schreiben
            SysFile.SysFileWrite(RTS_IEC_HANDLE_Ini,ADR(stHtmlDownload),TO_DWORD(LEN(stHtmlDownload)),ADR(RTS_IEC_RESULT_Ini));                                                                                                    
            stHtmlDownload  := '';      
            stHtmlDownload  := '</BODY></HTML>';                                                     
            // Daten Schreiben
            SysFile.SysFileWrite(RTS_IEC_HANDLE_Ini,ADR(stHtmlDownload),TO_DWORD(LEN(stHtmlDownload)),ADR(RTS_IEC_RESULT_Ini));                                                 
            SysFile.SysFileClose(RTS_IEC_HANDLE_Ini);   
        (* ID-Download *)    
            stFileDownloadHtml  :=  '';
            stFileDownloadHtml  :=  './visu/History/IDDownload.htm';                
            RTS_IEC_HANDLE_Ini := SysFile.SysFileOpen(stFileDownloadHtml,SysFile.ACCESS_MODE.AM_APPEND_PLUS,ADR(RTS_IEC_RESULT_Ini));
            // Schreibe Position festlegen
            SysFile.SysFileSetPos(RTS_IEC_HANDLE_Ini,0); 
            stHtmlDownload  := '';      
            stHtmlDownload  := '<HTML><HEAD><TITLE></TITLE></HEAD><BODY>';
            // Daten Schreiben
            SysFile.SysFileWrite(RTS_IEC_HANDLE_Ini,ADR(stHtmlDownload),TO_DWORD(LEN(stHtmlDownload)),ADR(RTS_IEC_RESULT_Ini));           
            stHtmlDownload  := '';      
            stHtmlDownload  := '<a href="Export/E_ID.csv" download = "E_ID.csv">E-ID Download</a><br />';                                                     
            // Daten Schreiben
            SysFile.SysFileWrite(RTS_IEC_HANDLE_Ini,ADR(stHtmlDownload),TO_DWORD(LEN(stHtmlDownload)),ADR(RTS_IEC_RESULT_Ini)); 
            stHtmlDownload  := '';      
            stHtmlDownload  := '<a href="Export/W_ID.csv" download = "W_ID.csv">W-ID Download</a><br />';                                                     
            // Daten Schreiben
            SysFile.SysFileWrite(RTS_IEC_HANDLE_Ini,ADR(stHtmlDownload),TO_DWORD(LEN(stHtmlDownload)),ADR(RTS_IEC_RESULT_Ini));                                                        
            stHtmlDownload  := '';      
            stHtmlDownload  := '<a href="Export/I_ID.csv" download = "I_ID.csv">I-ID Download</a><br />';                                                     
            // Daten Schreiben
            SysFile.SysFileWrite(RTS_IEC_HANDLE_Ini,ADR(stHtmlDownload),TO_DWORD(LEN(stHtmlDownload)),ADR(RTS_IEC_RESULT_Ini));                 
            stHtmlDownload  := '';      
            stHtmlDownload  := '</BODY></HTML>';                                                     
            // Daten Schreiben
            SysFile.SysFileWrite(RTS_IEC_HANDLE_Ini,ADR(stHtmlDownload),TO_DWORD(LEN(stHtmlDownload)),ADR(RTS_IEC_RESULT_Ini));                                                 
            SysFile.SysFileClose(RTS_IEC_HANDLE_Ini);                  
           RTS_IEC_HANDLE_Ini := 0;
            stFileDownloadHtml  :=  '';
            stFileDownloadHtml  :=  'History/HistoryDownload.htm';
        END_IF;        
        // Header erzeugen   
        metCreateHeader();
        // File öffnen
        metOpenFile(); 

    IF xIsNotSimulation THEN
            stFilePathDelete := '';
            stFilePathDelete := './visu/History/Export/E_ID.csv';
            SysFile.SysFileDelete(stFilePathDelete);
            stFilePathDelete := '';
            stFilePathDelete := './visu/History/Export/W_ID.csv';
            SysFile.SysFileDelete(stFilePathDelete);
            stFilePathDelete := '';            
            stFilePathDelete := './visu/History/Export/I_ID.csv';    
            SysFile.SysFileDelete(stFilePathDelete);        
    ELSE
            stFilePathDelete := '';
            stFilePathDelete := 'C:/PFC_Simulation/visu/History/Export/E_ID.csv';
            SysFile.SysFileDelete(stFilePathDelete);
            stFilePathDelete := '';
            stFilePathDelete := 'C:/PFC_Simulation/visu/History/Export/W_ID.csv';
            SysFile.SysFileDelete(stFilePathDelete);
            stFilePathDelete := '';
            stFilePathDelete := 'C:/PFC_Simulation/visu/History/Export/I_ID.csv';  
            SysFile.SysFileDelete(stFilePathDelete);
    END_IF;  
    udiSizeOfFileOnInit := TO_UDINT(SysFile.SysFileGetSize(stFilePathHistory,ADR(RTS_IEC_RESULT_Csv)));
    xInitDone := TRUE;
	__CATCH
		xInitDone := TRUE;
	__ENDTRY
END_IF;
END_ACTION

METHOD metReadCsv : BOOL
VAR_INPUT
    ITF_REPORTOBJECT_IN         :   ITF_REPORTOBJECT;
    diNr                        :   DINT;
END_VAR
VAR
    ITF_REPORTOBJECT_QUERY      :   ITF_REPORTOBJECT;
    stTemp                      :   STRING[255];
    dwPosRead                   :   DWORD;
    wFor                        :   WORD;
    diPosReadIst                :   DINT;
    dwBytesRead                 :   DWORD;
    scReportMetaData            :   scReportMetaData;
	pstDataToRead       		:   POINTER TO STRING[wSize];
	dwOldValue				: DWORD;
	ltStart					: LTIME;
	ltSafety				: LTIME; 
END_VAR
metReadCsv := FALSE;
IF __QUERYINTERFACE(ITF_REPORTOBJECT_IN,ITF_REPORTOBJECT_QUERY) AND_THEN diNr >= 1 AND diNr <= TO_DINT(proGetCountsOfReports) THEN
	pstDataToRead := __NEW(STRING[wSize]);
	IF pstDataToRead <> 0 THEN  
		pstDataToRead^ := '';
		metOpenFile();     
		dwPosRead := TO_DWORD((diNr -1 ) * wSize + wSizeHeader  +1);
		IF dwPosRead >= wSizeHeader AND dwPosRead > 0 AND RTS_IEC_HANDLE_Csv <> 0 THEN
			RTS_IEC_RESULT_Csv := SysFile.SysFileSetPos(RTS_IEC_HANDLE_Csv,TO_DWORD(dwPosRead));
			dwBytesRead := TO_DWORD(SysFile.SysFileRead(hFile:= RTS_IEC_HANDLE_Csv,pbyBuffer := pstDataToRead,ulSize := TO_DWORD(wSize-1),pResult := ADR(RTS_IEC_RESULT_Csv)));
			IF dwBytesRead = 0 THEN
				RETURN;
			END_IF;
			//get Data
			stTemp := '';
			FOR wFor := 0 TO MAX(wSize,1) -1 DO
				// Type
				IF wFor <= 6 THEN        
					stTemp[wFor]    := pstDataToRead^[wFor];
					stTemp[wFor+1]  := 0;
					IF wFor = 6 THEN
						IF FIND(stTemp,'ERROR') > 0 THEN
							scReportMetaData.enReportType := enReportType.Error;    
						ELSIF FIND(stTemp,'WARNING') > 0 THEN 
							scReportMetaData.enReportType := enReportType.Warning;  
						ELSIF FIND(stTemp,'INFO') > 0 THEN 
							scReportMetaData.enReportType := enReportType.Info;  
						END_IF
						stTemp := '';
					END_IF;
					CONTINUE;
				END_IF;
				// ID-Code
				IF wFor >= 8 AND wFor <= 17 THEN        
					stTemp[wFor-8]    := pstDataToRead^[wFor];
					stTemp[wFor-8+1]  := 0;
					IF wFor = 17 THEN
						StrTrimA(ADR(stTemp));
						scReportMetaData.uliReportId := TO_ULINT(stTemp);
						stTemp := '';
					END_IF;
					CONTINUE;
				END_IF;                  
				// Dt From              
				IF wFor >= 311 AND wFor <= 332 THEN        
					stTemp[wFor-311]    := pstDataToRead^[wFor];
					stTemp[wFor-311+1]  := 0;
					IF wFor = 332 THEN
						StrTrimA(ADR(stTemp));
						scReportMetaData.dtFrom := TO_DT(stTemp);
						stTemp := '';
					END_IF;
				END_IF;
				// Dt To
				IF wFor >= 334 AND wFor <= 355 THEN        
					stTemp[wFor-334]    := pstDataToRead^[wFor];
					stTemp[wFor-334+1]  := 0;
					IF wFor = 355 THEN
						StrTrimA(ADR(stTemp));
						scReportMetaData.dtTo := TO_DT(stTemp);
						IF scReportMetaData.dtTo = TO_DT(0) AND diNr <= proGetCountOfReportsOnInit THEN
							scReportMetaData.dtTo := scReportMetaData.dtFrom;
						END_IF
						stTemp := '';
					END_IF;
					CONTINUE;
				END_IF;  
				// Is Quitt
				IF wFor >= 357 AND wFor <= 361 THEN        
					stTemp[wFor-357]    := pstDataToRead^[wFor];
					stTemp[wFor-357+1]  := 0;
					IF wFor = 361 THEN
						StrTrimA(ADR(stTemp));
						IF diNr > proGetCountOfReportsOnInit THEN
							scReportMetaData.xIsQuitt := TO_BOOL(stTemp);
						ELSE
							scReportMetaData.xIsQuitt := TRUE;
						END_IF;                        
						stTemp := '';
					END_IF;
					CONTINUE;
				END_IF;                 
				// Report Text List
				IF wFor >= 363 AND wFor <= 462 THEN        
					stTemp[wFor-363]    := pstDataToRead^[wFor];
					stTemp[wFor-363+1]  := 0;
					IF wFor = 462 THEN
						StrTrimA(ADR(stTemp));
						scReportMetaData.stReportTextList := LEFT(stTemp,100);
						stTemp := '';
					END_IF;
					CONTINUE;
				END_IF;  
				// Report Text List Id
				IF wFor >= 464 AND wFor <= 466 THEN        
					stTemp[wFor-464]    := pstDataToRead^[wFor];
					stTemp[wFor-464+1]  := 0;
					IF wFor = 466 THEN
						StrTrimA(ADR(stTemp));
						scReportMetaData.stReportTxtId := LEFT(stTemp,3);
						stTemp := '';
					END_IF;
				END_IF;  
				// Report Acknowledg Type
				IF wFor >= 468 AND wFor <= 470 THEN        
					stTemp[wFor-468]    := pstDataToRead^[wFor];
					stTemp[wFor-468+1]  := 0;
					IF wFor = 470 THEN
						scReportMetaData.enReportacknowledgeType := TO_INT(stTemp);
						stTemp := '';
					END_IF;
					CONTINUE;
				END_IF;          
				// Object Id
				IF wFor >= 472 AND wFor <= 491 THEN        
					stTemp[wFor-472]    := pstDataToRead^[wFor];
					stTemp[wFor-472+1]  := 0;
					IF wFor = 491 THEN
						StrTrimA(ADR(stTemp));
						ITF_REPORTOBJECT_QUERY.proReporterObjectId := LEFT(stTemp,20);
						stTemp := '';
					END_IF;
					CONTINUE;
				END_IF;      
				// Instance Path
				IF wFor >= 493 AND wFor <= 747 THEN        
					stTemp[wFor-493]    := pstDataToRead^[wFor];
					stTemp[wFor-493+1]  := 0;
					IF wFor = 747 THEN
						StrTrimA(ADR(stTemp));
						ITF_REPORTOBJECT_QUERY.proSetInstancePath := stTemp;
						stTemp := '';
					END_IF;
					CONTINUE;
				END_IF;      
				// Additional Text
				IF wFor >= 749 AND wFor <= 768 THEN        
					stTemp[wFor-749]    := pstDataToRead^[wFor];
					stTemp[wFor-749+1]  := 0;
					IF wFor = 768 THEN
						StrTrimA(ADR(stTemp));
						scReportMetaData.stAdditionalText := LEFT(stTemp,20);
						stTemp := '';
					END_IF;
					CONTINUE;
				END_IF; 
				// Prio
				IF wFor >= 770 AND wFor <= 772 THEN        
					stTemp[wFor-770]    := pstDataToRead^[wFor];
					stTemp[wFor-770+1]  := 0;
					IF wFor = 772 THEN
						StrTrimA(ADR(stTemp));
						scReportMetaData.usiPrio := TO_USINT(LEFT(stTemp,3));
						stTemp := '';
					END_IF;
					CONTINUE;
				END_IF;           
				// Report In
				IF wFor >= 774 AND wFor <= 778 THEN        
					stTemp[wFor-774]    := pstDataToRead^[wFor];
					stTemp[wFor-774+1]  := 0;
					IF wFor = 778 THEN
						StrTrimA(ADR(stTemp));
						IF diNr > proGetCountOfReportsOnInit THEN
							scReportMetaData.xReportIn := TO_BOOL(LEFT(stTemp,5));
						ELSE
							scReportMetaData.xReportIn := FALSE;
						END_IF;
						stTemp := '';
					END_IF;
				END_IF;        
				// State
				IF wFor >= 780 AND wFor <= 784 THEN        
					stTemp[wFor-780]    := pstDataToRead^[wFor];
					stTemp[wFor-780+1]  := 0;
					IF wFor = 784 THEN
						StrTrimA(ADR(stTemp));
						IF diNr > proGetCountOfReportsOnInit THEN
							scReportMetaData.xActive   := TO_BOOL(LEFT(stTemp,5));
						ELSE
							scReportMetaData.xActive := FALSE;
						END_IF;
						stTemp := '';
						ITF_REPORTOBJECT_QUERY.proSetMetaData := scReportMetaData;
						metReadCsv := TRUE;
					END_IF;
				END_IF;             
			END_FOR;
		END_IF;
	END_IF;      
	__DELETE(pstDataToRead);  
END_IF;
END_METHOD

PROPERTY proGetCountsOfReports : UDINT
GET
proGetCountsOfReports := 0;
__TRY
	udiSizeOfFileNow := TO_UDINT(SysFile.SysFileGetSizeByHandle(RTS_IEC_HANDLE_Csv,ADR(RTS_IEC_RESULT_Csv)));
	IF wSize > 0 THEN
		proGetCountsOfReports := (udiSizeOfFileNow - TO_UDINT(SIZEOF(stHeader)-1))/TO_UDINT(wSize);
		udiOldValueCounts := proGetCountsOfReports;
	END_IF;	
__CATCH
	proGetCountsOfReports := udiOldValueCounts;	
__ENDTRY
END_GET
END_PROPERTY

PROPERTY proGetCountOfReportsOnInit : INT
GET
IF wSize > 0 THEN
    proGetCountOfReportsOnInit := TO_INT((udiSizeOfFileOnInit - TO_UDINT(SIZEOF(stHeader)-1))/TO_UDINT(wSize));
END_IF;
END_GET
END_PROPERTY

METHOD metCreateHeader : BOOL
VAR_INPUT
END_VAR
IF RTS_IEC_HANDLE_Csv = 0 THEN
    udiSizeOfFileNow := TO_UDINT(SysFile.SysFileGetSize(stFilePathHistory,ADR(RTS_IEC_RESULT_Csv))); 
    IF udiSizeOfFileNow = 0 THEN
        RTS_IEC_HANDLE_Csv := SysFile.SysFileOpen(stFilePathHistory,SysFile.ACCESS_MODE.AM_APPEND_PLUS,ADR(RTS_IEC_RESULT_Csv));
        // Schreibe Position festlegen
        SysFile.SysFileSetPos(RTS_IEC_HANDLE_Csv,0);  
        stHeader  := '';      
        stHeader  := 'Type;ID;Object-Name;Reporttext;DT-From;DT-To;Is-Quitt;Report TextList;Text-ID;Type of Acknowledg;Object-Id;Instance-Path;Additional-Text;Prio;In;State';
        stHeader[wSizeHeader] := stRN[0];
        // Daten Schreiben
        SysFile.SysFileWrite(RTS_IEC_HANDLE_Csv,ADR(stHeader),SIZEOF(stHeader),ADR(RTS_IEC_RESULT_Csv));        
        SysFile.SysFileClose(RTS_IEC_HANDLE_Csv);
        RTS_IEC_HANDLE_Csv := 0;
    END_IF;
END_IF;
END_METHOD

PROPERTY proExportIdStart : BOOL
SET
VAR
    stTemp  :   STRING(255);
END_VAR
IF proExportIdStart AND NOT xExportId THEN
    xExportId := TRUE;
    stTemp    := '';
    stTemp    := './visu/History/Export/E_ID.csv';
    RTS_IEC_HANDLE_ExE := SysFile.SysFileOpen(stTemp,ACCESS_MODE.AM_WRITE_PLUS,ADR(RTS_IEC_RESULT_Exp));
    stTemp    := '';
    stTemp    := './visu/History/Export/W_ID.csv';
    RTS_IEC_HANDLE_ExW := SysFile.SysFileOpen(stTemp,ACCESS_MODE.AM_WRITE_PLUS,ADR(RTS_IEC_RESULT_Exp));
    stTemp    := '';
    stTemp    := './visu/History/Export/I_ID.csv';
    RTS_IEC_HANDLE_ExI := SysFile.SysFileOpen(stTemp,ACCESS_MODE.AM_WRITE_PLUS,ADR(RTS_IEC_RESULT_Exp));    
    stTemp    := '';
    stTemp    := 'REPORT TYPE;ID;BMK;AKS;VENDOR DESIGNATION;REPORT TEXT$R';
    SysFile.SysFileWrite(RTS_IEC_HANDLE_ExE,ADR(stTemp),TO_UINT(LEN(stTemp)),ADR(RTS_IEC_RESULT_Exp));    
    SysFile.SysFileWrite(RTS_IEC_HANDLE_ExW,ADR(stTemp),TO_UINT(LEN(stTemp)),ADR(RTS_IEC_RESULT_Exp));
    SysFile.SysFileWrite(RTS_IEC_HANDLE_ExI,ADR(stTemp),TO_UINT(LEN(stTemp)),ADR(RTS_IEC_RESULT_Exp));   
END_IF
END_SET
GET
proExportIdStart := xExportId;
END_GET
END_PROPERTY

METHOD metExportId : BOOL
VAR_INPUT
    ITF_BMK_IN                  :   CtaAppBmk.ITF_BMK;
    stReportTextListIn          :   stReportTextList;
    iId                         :   INT;
    enReportTypeIn      		:   enReportType;
    enReportAcknowledgeTypeIn   :   enReportAcknowledgeType;    
END_VAR
VAR
    stTemp                      :   STRING(255);
    stId                        :   STRING(3);
    ITF_BMK_QUERY               :   CtaAppBmk.ITF_BMK;     
    RTS_IEC_HANDLE_Exp          :   RTS_IEC_HANDLE;
    diIndex                     :   DINT;
END_VAR
IF ITF_BMK_NEXT_EXPORT = ITF_BMK_IN THEN
    ITF_BMK_NEXT_EXPORT := 0;
    diIndex :=__XADD(ADR(diCountExp),-diCountExp);
END_IF;
diIndex :=__XADD(ADR(diCountExp),1);
IF diIndex <= Parameter.diMaxExportsPerCycle THEN
    xIsExporting := TRUE;
    (* Type of Report *)
    stTemp := '';
    IF enReportTypeIn = enReportType.Error THEN
        stTemp := 'ERROR';
        RTS_IEC_HANDLE_Exp  := RTS_IEC_HANDLE_ExE;
    ELSIF enReportTypeIn = enReportType.Warning THEN
        stTemp := 'WARNING';
        RTS_IEC_HANDLE_Exp  := RTS_IEC_HANDLE_ExW;
    ELSIF enReportTypeIn = enReportType.Info THEN   
        stTemp := 'INFO';
        RTS_IEC_HANDLE_Exp  := RTS_IEC_HANDLE_ExI;
    END_IF;
    (* Check Handle *)    
    IF RTS_IEC_HANDLE_Exp <> 0 AND __QUERYINTERFACE(ITF_BMK_IN,ITF_BMK_QUERY) THEN
        (* Write Type *)
        SysFile.SysFileWrite(RTS_IEC_HANDLE_Exp,ADR(stTemp),TO_UINT(LEN(stTemp)),ADR(RTS_IEC_RESULT_Exp));
        (* Write Semicolon *)
        stTemp := '';
        stTemp := ';';
        SysFile.SysFileWrite(RTS_IEC_HANDLE_Exp,ADR(stTemp),TO_UINT(LEN(stTemp)),ADR(RTS_IEC_RESULT_Exp));
        (* Write ID *)
        stTemp := '';
        stTemp := TO_STRING(fcBmkToId(ITF_BMK_QUERY.proGetBMK,TO_DINT(iId),FALSE,enReportTypeIn));
        SysFile.SysFileWrite(RTS_IEC_HANDLE_Exp,ADR(stTemp),TO_UINT(LEN(stTemp)),ADR(RTS_IEC_RESULT_Exp));
        (* Write Semicolon *)
        stTemp := '';
        stTemp := ';';
        SysFile.SysFileWrite(RTS_IEC_HANDLE_Exp,ADR(stTemp),TO_UINT(LEN(stTemp)),ADR(RTS_IEC_RESULT_Exp));
        (* Write BMK *)
        stTemp := '';
        stTemp := ITF_BMK_QUERY.proGetBMK;
        SysFile.SysFileWrite(RTS_IEC_HANDLE_Exp,ADR(stTemp),TO_UINT(LEN(stTemp)),ADR(RTS_IEC_RESULT_Exp));
        (* Write Semicolon *)
        stTemp := '';
        stTemp := ';';
        SysFile.SysFileWrite(RTS_IEC_HANDLE_Exp,ADR(stTemp),TO_UINT(LEN(stTemp)),ADR(RTS_IEC_RESULT_Exp));    
        (* Write AKS *)
        stTemp := '';
        stTemp := ITF_BMK_QUERY.proGetAKS;
        SysFile.SysFileWrite(RTS_IEC_HANDLE_Exp,ADR(stTemp),TO_UINT(LEN(stTemp)),ADR(RTS_IEC_RESULT_Exp));
        (* Write Semicolon *)
        stTemp := '';
        stTemp := ';';
        SysFile.SysFileWrite(RTS_IEC_HANDLE_Exp,ADR(stTemp),TO_UINT(LEN(stTemp)),ADR(RTS_IEC_RESULT_Exp));        
        (* Write Vendordesignation*)
        stTemp := '';
        stTemp := ITF_BMK_QUERY.proGetVendorDesignation;
        IF stTemp = '' THEN
            stTemp := ITF_BMK_QUERY.proGetInstancePath;
		END_IF;
        SysFile.SysFileWrite(RTS_IEC_HANDLE_Exp,ADR(stTemp),TO_UINT(LEN(stTemp)),ADR(RTS_IEC_RESULT_Exp));
        (* Write Semicolon *)
        stTemp := '';
        stTemp := ';';
        SysFile.SysFileWrite(RTS_IEC_HANDLE_Exp,ADR(stTemp),TO_UINT(LEN(stTemp)),ADR(RTS_IEC_RESULT_Exp));    
        (* Write Report Text *)
        stTemp := '';
        (*Load Text By Language*)
        stId   := TO_STRING(iId);
        stTemp := CmpDynamicText.DynamicTextGetText(ADR(stReportTextListIn),ADR(stId))^;
        (* Load Default Text if no spezifig Language*)
        IF stTemp = '' THEN
            stTemp := CmpDynamicText.DynamicTextGetDefaultText(ADR(stReportTextListIn),ADR(stId))^;
        END_IF;
        SysFile.SysFileWrite(RTS_IEC_HANDLE_Exp,ADR(stTemp),TO_UINT(LEN(stTemp)),ADR(RTS_IEC_RESULT_Exp));
        (* Write $R *)
        stTemp := '';
        stTemp := '$R';
        SysFile.SysFileWrite(RTS_IEC_HANDLE_Exp,ADR(stTemp),TO_UINT(LEN(stTemp)),ADR(RTS_IEC_RESULT_Exp));        
        metExportId := TRUE;     
    END_IF;
ELSE
    IF ITF_BMK_NEXT_EXPORT = 0 THEN
        ITF_BMK_NEXT_EXPORT := ITF_BMK_IN;
    END_IF;    
END_IF;
END_METHOD

METHOD metResetCycleCount : BOOL
VAR_INPUT
END_VAR
IF xExportDoneTemp THEN
    iWait := iWait + 1;
END_IF;
IF xExportDoneTemp AND NOT xIsExporting AND iWait >= 500 THEN
    xExportDone         := TRUE;
    xExportDoneTemp     := FALSE;
    xExportId           := FALSE;
    ITF_BMK_NEXT_EXPORT := 0;
    diCountExp          := 0;
    IF RTS_IEC_HANDLE_ExE <> 0 THEN
        SysFile.SysFileClose(RTS_IEC_HANDLE_ExE);
        RTS_IEC_HANDLE_ExE  := 0;
    END_IF;
    IF RTS_IEC_HANDLE_ExW <> 0 THEN
        SysFile.SysFileClose(RTS_IEC_HANDLE_ExW);
        RTS_IEC_HANDLE_ExW  := 0;
    END_IF;
    IF RTS_IEC_HANDLE_ExI <> 0 THEN
        SysFile.SysFileClose(RTS_IEC_HANDLE_ExI);
        RTS_IEC_HANDLE_ExI  := 0;
    END_IF;    
END_IF;
IF xIsExporting THEN
    xExportDoneTemp := TRUE;
    xExportDone     := FALSE;
    xIsExporting    := FALSE;
    iWait           := 0;
END_IF;
END_METHOD

PROPERTY proExport : BOOL
GET
proExport := xExportId;
END_GET
END_PROPERTY

PROPERTY proIsRegistred : BOOL
SET
xIsRegistretAppEvent := proIsRegistred;
END_SET
GET
proIsRegistred := xIsRegistretAppEvent;
END_GET
END_PROPERTY

METHOD metStartDone : BOOL
RETURN;
END_METHOD

METHOD metPrepeareStop : BOOL
metCloseFile();
END_METHOD

PROPERTY proDenyStop : BOOL
GET
proDenyStop := NOT xInitDone;
END_GET
END_PROPERTY

METHOD metCyclicCall : BOOL
(* Reset CycleCount Csv *)
metResetCycleCount();
END_METHOD

METHOD PRIVATE metWriteOnChange : BOOL
VAR_INPUT
    ITF_REPORTOBJECT_IN 	: ITF_REPORTOBJECT;
    dwWritePos   			:   DWORD;
END_VAR
VAR
    ITF_REPORTOBJECT_QUERY  :   ITF_REPORTOBJECT;
    stTemp         	 		:   STRING[255];
    dwIstPso        		:   DWORD;
	pstDataToWriteT     	:   POINTER TO STRING[wSize]; 
	diFor               :   DINT;
END_VAR
IF __QUERYINTERFACE(ITF_REPORTOBJECT_IN,ITF_REPORTOBJECT_QUERY) AND wSize <> 0 THEN
    pstDataToWriteT := __NEW(STRING[wSize]);
    IF pstDataToWriteT <> 0 THEN    
        // Daten zum Schreiben erzeugen
        pstDataToWriteT^  :=    '';
        stTemp := '';
        IF ITF_REPORTOBJECT_QUERY.proReportType = enReportType.Error THEN
            stTemp := 'ERROR';
        ELSIF ITF_REPORTOBJECT_QUERY.proReportType = enReportType.Warning THEN
            stTemp := 'WARNING';
        ELSIF ITF_REPORTOBJECT_QUERY.proReportType = enReportType.Info THEN
            stTemp := 'INFO';
        END_IF;
        metFillSpace(stTemp,7);
        StrConcatA(ADR(stTemp),pstDataToWriteT,TO_INT(SIZEOF(pstDataToWriteT^)));  
        stTemp := '';
        stTemp := stSC;
        StrConcatA(ADR(stTemp),pstDataToWriteT,TO_INT(SIZEOF(pstDataToWriteT^)));     
        stTemp := '';
        stTemp := TO_STRING(ITF_REPORTOBJECT_QUERY.proReportId);
        metFillSpace(stTemp,10);
        StrConcatA(ADR(stTemp),pstDataToWriteT,TO_INT(SIZEOF(pstDataToWriteT^)));    
        stTemp := '';
        stTemp := stSC;
        StrConcatA(ADR(stTemp),pstDataToWriteT,TO_INT(SIZEOF(pstDataToWriteT^)));                    
        stTemp := '';
        stTemp := TO_STRING(ITF_REPORTOBJECT_QUERY.proGetReporterText);
        metFillSpace(stTemp,150);
        StrConcatA(ADR(stTemp),pstDataToWriteT,TO_INT(SIZEOF(pstDataToWriteT^)));                                        
        stTemp := '';
        stTemp := stSC;
        StrConcatA(ADR(stTemp),pstDataToWriteT,TO_INT(SIZEOF(pstDataToWriteT^)));
        stTemp := '';
        stTemp := TO_STRING(ITF_REPORTOBJECT_QUERY.proGetReportText);
        metFillSpace(stTemp,140); 
        StrConcatA(ADR(stTemp),pstDataToWriteT,TO_INT(SIZEOF(pstDataToWriteT^)));               
        stTemp := '';
        stTemp := stSC;
        StrConcatA(ADR(stTemp),pstDataToWriteT,TO_INT(SIZEOF(pstDataToWriteT^)));        
        stTemp := '';
        stTemp := TO_STRING(ITF_REPORTOBJECT_QUERY.proDtFrom);
        metFillSpace(stTemp,22);
        StrConcatA(ADR(stTemp),pstDataToWriteT,TO_INT(SIZEOF(pstDataToWriteT^)));  
        stTemp := '';
        stTemp := stSC;
        StrConcatA(ADR(stTemp),pstDataToWriteT,TO_INT(SIZEOF(pstDataToWriteT^)));
        stTemp := '';
        stTemp := TO_STRING(ITF_REPORTOBJECT_QUERY.proDtTo); 
        metFillSpace(stTemp,22);
        StrConcatA(ADR(stTemp),pstDataToWriteT,TO_INT(SIZEOF(pstDataToWriteT^))); 
        stTemp := '';
        stTemp := stSC;
        StrConcatA(ADR(stTemp),pstDataToWriteT,TO_INT(SIZEOF(pstDataToWriteT^)));
        stTemp := '';
        stTemp := TO_STRING(ITF_REPORTOBJECT_QUERY.proIsQuitt);
        metFillSpace(stTemp,5);
        StrConcatA(ADR(stTemp),pstDataToWriteT,TO_INT(SIZEOF(pstDataToWriteT^))); 
        stTemp := '';
        stTemp := stSC;
        StrConcatA(ADR(stTemp),pstDataToWriteT,TO_INT(SIZEOF(pstDataToWriteT^)));
        stTemp := '';
        stTemp := TO_STRING(ITF_REPORTOBJECT_QUERY.proReportTextList);
        metFillSpace(stTemp,100);
        StrConcatA(ADR(stTemp),pstDataToWriteT,TO_INT(SIZEOF(pstDataToWriteT^))); 
        stTemp := '';
        stTemp := stSC;
        StrConcatA(ADR(stTemp),pstDataToWriteT,TO_INT(SIZEOF(pstDataToWriteT^)));
        stTemp := '';
        stTemp := TO_STRING(ITF_REPORTOBJECT_QUERY.proReportTextId);
        metFillSpace(stTemp,3);
        StrConcatA(ADR(stTemp),pstDataToWriteT,TO_INT(SIZEOF(pstDataToWriteT^)));                       
        stTemp := '';
        stTemp := stSC;
        StrConcatA(ADR(stTemp),pstDataToWriteT,TO_INT(SIZEOF(pstDataToWriteT^)));
        stTemp := '';
        stTemp := TO_STRING(TO_USINT(ITF_REPORTOBJECT_QUERY.proReportAcknowledgType));
        metFillSpace(stTemp,3);
        StrConcatA(ADR(stTemp),pstDataToWriteT,TO_INT(SIZEOF(pstDataToWriteT^)));
        stTemp := '';
        stTemp := stSC;
        StrConcatA(ADR(stTemp),pstDataToWriteT,TO_INT(SIZEOF(pstDataToWriteT^)));
        stTemp := '';
        stTemp := ITF_REPORTOBJECT_QUERY.proGetObjectId;
        metFillSpace(stTemp,20);        
        StrConcatA(ADR(stTemp),pstDataToWriteT,TO_INT(SIZEOF(pstDataToWriteT^))); 
        stTemp := '';
        stTemp := stSC;
        StrConcatA(ADR(stTemp),pstDataToWriteT,TO_INT(SIZEOF(pstDataToWriteT^)));
        stTemp := '';
        stTemp := ITF_REPORTOBJECT_QUERY.proGetInstancePath;
        metFillSpace(stTemp,255);      
        StrConcatA(ADR(stTemp),pstDataToWriteT,TO_INT(SIZEOF(pstDataToWriteT^)));
        stTemp := '';
        stTemp := stSC;
        StrConcatA(ADR(stTemp),pstDataToWriteT,TO_INT(SIZEOF(pstDataToWriteT^)));
        stTemp := '';
        stTemp := ITF_REPORTOBJECT_QUERY.proAdditionalText;
        metFillSpace(stTemp,20);
        StrConcatA(ADR(stTemp),pstDataToWriteT,TO_INT(SIZEOF(pstDataToWriteT^)));
        stTemp := '';
        stTemp := stSC;
        StrConcatA(ADR(stTemp),pstDataToWriteT,TO_INT(SIZEOF(pstDataToWriteT^)));            
        stTemp := '';
        stTemp := TO_STRING(ITF_REPORTOBJECT_QUERY.proPrio);
        metFillSpace(stTemp,3); 
        StrConcatA(ADR(stTemp),pstDataToWriteT,TO_INT(SIZEOF(pstDataToWriteT^)));      
        stTemp := '';
        stTemp := stSC;
        StrConcatA(ADR(stTemp),pstDataToWriteT,TO_INT(SIZEOF(pstDataToWriteT^)));
        stTemp := '';
        stTemp := TO_STRING(ITF_REPORTOBJECT_QUERY.proReportIn);
        metFillSpace(stTemp,5);                
        StrConcatA(ADR(stTemp),pstDataToWriteT,TO_INT(SIZEOF(pstDataToWriteT^))); 
        stTemp := '';
        stTemp := stSC;
        StrConcatA(ADR(stTemp),pstDataToWriteT,TO_INT(SIZEOF(pstDataToWriteT^)));
        stTemp := '';
        stTemp := TO_STRING(ITF_REPORTOBJECT_QUERY.proStateActive);
        metFillSpace(stTemp,5);                
        StrConcatA(ADR(stTemp),pstDataToWriteT,TO_INT(SIZEOF(pstDataToWriteT^)));         
        (* String mit Lehrzeichen auffüllen und mit $R abschliessen *)                     
        FOR diFor := StrLenA(pstDataToWriteT) TO wSize -1 DO
            IF diFor < wSize -1 THEN
                pstDataToWriteT^[diFor] := stSpace[0];
            ELSE
                pstDataToWriteT^[diFor] := stRN[0];
            END_IF;
        END_FOR;                          
        // Daten Schreiben
        IF metOpenFile() THEN
            SysFile.SysFileSetPos(RTS_IEC_HANDLE_Csv,dwWritePos);
            SysFile.SysFileGetPos(RTS_IEC_HANDLE_Csv,ADR(dwIstPso));        
			IF dwWritePos = dwIstPso THEN   
            	dwWrite := TO_DWORD(SysFile.SysFileWrite(RTS_IEC_HANDLE_Csv,pstDataToWriteT,SIZEOF(pstDataToWriteT^)-1,ADR(RTS_IEC_RESULT_Csv)));
			END_IF;	
        END_IF;
        __DELETE(pstDataToWriteT);
    END_IF;
END_IF;
END_METHOD

METHOD metDeleteHistory : BOOL
VAR_INPUT
END_VAR
IF RTS_IEC_HANDLE_Csv = 0 THEN
    RTS_IEC_RESULT_Csv := SysFile.SysFileDelete(stFilePathHistory);
ELSE
    RTS_IEC_RESULT_Csv := SysFile.SysFileClose(RTS_IEC_HANDLE_Csv);
    RTS_IEC_HANDLE_Csv := 0;
    IF RTS_IEC_RESULT_Csv = 0 THEN
        RTS_IEC_RESULT_Csv := SysFile.SysFileDelete(stFilePathHistory); 
    END_IF;
END_IF
IF RTS_IEC_RESULT_Csv = 0 THEN
    metCreateHeader();
    udiSizeOfFileOnInit := TO_UDINT(SysFile.SysFileGetSize(stFilePathHistory,ADR(RTS_IEC_RESULT_Csv)));
    udiSizeOfFileNow    := udiSizeOfFileOnInit;
    GVL_Report.fbReportObjectFactory.metReSaveAfterDelete();
    GVL_Report.fbReportVisu.proOffset := 0;
    GVL_Report.fbReportVisu.metReload();
END_IF;
END_METHOD

METHOD metAddObjForeWriteDtFrom
VAR_INPUT
	ITF_REPORTOBJECT_IN 	: ITF_REPORTOBJECT;	
END_VAR
VAR
	diOldValue				: DINT;
END_VAR
IF __QUERYINTERFACE(ITF_REPORTOBJECT_IN,ITF_REPORTOBJECT_IN) THEN
		diOldValue	:= __XADD(ADR(diNextFreeDtFrom),1);	
		IF diOldValue >= LOWER_BOUND(ayITF_WriteDtFrom,1) AND diOldValue <= UPPER_BOUND(ayITF_WriteDtFrom,1) THEN
			ayITF_WriteDtFrom[diOldValue] := ITF_REPORTOBJECT_IN;
		END_IF;
END_IF;
END_METHOD

METHOD metAddObjForeWriteDtTo
VAR_INPUT
	ITF_REPORTOBJECT_IN 	: ITF_REPORTOBJECT;	
END_VAR
VAR
	diOldValue				: DINT;
END_VAR
IF __QUERYINTERFACE(ITF_REPORTOBJECT_IN,ITF_REPORTOBJECT_IN) THEN
	IF ITF_REPORTOBJECT_IN.proWritePosInCsv > 0 THEN
		diOldValue	:= __XADD(ADR(diNextFreeDtTo),1);	
		IF diOldValue >= LOWER_BOUND(ayITF_WriteDtTo,1) AND diOldValue <= UPPER_BOUND(ayITF_WriteDtTo,1) THEN
			ayITF_WriteDtTo[diOldValue] := ITF_REPORTOBJECT_IN;
		END_IF;
	END_IF;
END_IF;
END_METHOD

METHOD metAddObjForeWriteOnChange
VAR_INPUT
	ITF_REPORTOBJECT_IN 	: ITF_REPORTOBJECT;	
END_VAR
VAR
	diOldValue				: DINT;
END_VAR
IF __QUERYINTERFACE(ITF_REPORTOBJECT_IN,ITF_REPORTOBJECT_IN) THEN
	IF ITF_REPORTOBJECT_IN.proWritePosInCsv > 0 THEN
		diOldValue	:= __XADD(ADR(diNextFreeChange),1);	
		IF diOldValue >= LOWER_BOUND(ayITF_WriteChange,1) AND diOldValue <= UPPER_BOUND(ayITF_WriteChange,1) THEN
			ayITF_WriteChange[diOldValue] := ITF_REPORTOBJECT_IN;
		END_IF;
	END_IF;	
END_IF;
END_METHOD

END_FUNCTION_BLOCK

// 21 Interface/ITF_REPORTOBJECT
INTERFACE ITF_REPORTOBJECT EXTENDS CtaAppBmk.ITF_BMK;

PROPERTY FINAL proGetReportText : STRING[140]
GET
END_GET
END_PROPERTY

PROPERTY FINAL proStateActive : BOOL
SET
END_SET
GET
END_GET
END_PROPERTY

PROPERTY FINAL proIsQuitt : BOOL
SET
END_SET
GET
END_GET
END_PROPERTY

PROPERTY FINAL proIsSelected : BOOL
SET
END_SET
GET
END_GET
END_PROPERTY

PROPERTY FINAL proReportId : ULINT
GET
END_GET
END_PROPERTY

PROPERTY FINAL proMaxRetry : INT
SET
END_SET
GET
END_GET
END_PROPERTY

PROPERTY FINAL proCountRetry : INT
SET
END_SET
GET
END_GET
END_PROPERTY

PROPERTY FINAL proReportTextList : STRING[100]
SET
END_SET
GET
END_GET
END_PROPERTY

PROPERTY FINAL proReportTextId : STRING[3]
SET
END_SET
GET
END_GET
END_PROPERTY

PROPERTY FINAL proReporterObjectId : STRING[20]
SET
END_SET
GET
END_GET
END_PROPERTY

PROPERTY FINAL proAdditionalText : STRING(20)
SET
END_SET
GET
END_GET
END_PROPERTY

PROPERTY FINAL proReportType : enReportType
SET
END_SET
GET
END_GET
END_PROPERTY

PROPERTY FINAL proReportAcknowledgType : enReportacknowledgeType
SET
END_SET
GET
END_GET
END_PROPERTY

PROPERTY FINAL proWritePosInCsv : DWORD
SET
END_SET
GET
END_GET
END_PROPERTY

PROPERTY FINAL proGetReporterText : STRING[150]
GET
END_GET
END_PROPERTY

PROPERTY FINAL proReportIn : BOOL
SET
END_SET
GET
END_GET
END_PROPERTY

PROPERTY FINAL proDtTo : DT
SET
END_SET
GET
END_GET
END_PROPERTY

PROPERTY FINAL proDtFrom : DT
SET
END_SET
GET
END_GET
END_PROPERTY

METHOD FINAL metReportObject : BOOL
VAR_INPUT
END_VAR
END_METHOD

PROPERTY FINAL proQuitt : BOOL
SET
END_SET
GET
END_GET
END_PROPERTY

PROPERTY FINAL proSetMetaData : scReportMetaData
SET
END_SET
END_PROPERTY

PROPERTY FINAL proPrio : USINT
SET
END_SET
GET
END_GET
END_PROPERTY

METHOD FINAL metDestroy
VAR_INPUT
END_VAR
END_METHOD

METHOD FINAL metWriteDtFromToCsv : DWORD
VAR_INPUT
END_VAR
END_METHOD

METHOD FINAL metSaveOnChange : BOOL
VAR_INPUT
END_VAR
END_METHOD

END_INTERFACE

// 30 Program Organization Units/fcBmkToId
FUNCTION fcBmkToId  :   ULINT;
VAR_INPUT
    stBMK           :   STRING             [8];                                                                     // BMK als STRING [8]
    diNr            :   DINT;                                                                                       // Nr welche am ende angefügt wird
    xNoZero         :   BOOL;                                                                                       // Bei 1-Stelliger Nummer keine 0 voransetzen
    enReportTypeIn  :   enReportType;
END_VAR
VAR
    iFor            :   INT;                                                                                        // Forschleifen Variable
    iOfset          :   INT;                                                                                        // Offsetvariable 
    pstBMK          :   POINTER TO STRING  [8];                                                                    // Pointer auf stBMK
    pstBmkAscii     :   POINTER TO STRING  [12];                                                                    // Pointer auf stBmkAscii
    stBmkAscii      :   STRING             [12];                                                                    // String mit dem Numerischen BMK Code
    iAkt            :   INT;
END_VAR

//===========================================================================================================================================================================================================================================//
//  Pointer zuweisung		                                                                          																															             //
//===========================================================================================================================================================================================================================================// 
pstBMK          := ADR(stBMK);
pstBmkAscii     := ADR(stBmkAscii);
pstBmkAscii^[0] := STRING_TO_BYTE('');      // Pointer Cleaning Byte 0

IF pstBMK <> 0 AND pstBmkAscii <> 0 AND StBMK <> '' THEN
    //===========================================================================================================================================================================================================================================//
    //  BMK TO DINT Wandeln		                                                                          																															             //
    //===========================================================================================================================================================================================================================================// 
    FOR iFor := 0 TO LEN(stBMK) BY 1 DO
        iAkt    :=  BYTE_TO_INT(pstBMK^[iFor]);
        pstBmkAscii^[iFor + iOfset + 1] := STRING_TO_BYTE('');                                                          // Byte in Pointer Cleanen 
        IF BYTE_TO_INT(pstBMK^[iFor])>= 48 AND BYTE_TO_INT(pstBMK^[iFor]) <= 57 THEN                                    // ASCII Zahlen von 48 bis 57 = 0 bis 9
            pstBmkAscii^[iFor + iOfset] := pstBMK^[iFor];
        ELSIF BYTE_TO_INT(pstBMK^[iFor])>= 65 AND BYTE_TO_INT(pstBMK^[iFor]) <= 90 THEN                                 // ASCII Grosbuchstaben von 65 bis 90 = A bis Z
            pstBmkAscii^                := CONCAT(pstBmkAscii^,INT_TO_STRING(BYTE_TO_INT(pstBMK^[iFor])));
            iOfset                      := iOfset + 1;                                                                  // Zeichenversatz von + 1 je buchstaben 
        ELSIF BYTE_TO_INT(pstBMK^[iFor])>= 97 AND BYTE_TO_INT(pstBMK^[iFor]) <= 120 THEN                                // ASCII kleinbuchstaben von 97 bis 120 = a bis z 
            pstBmkAscii^                := CONCAT(pstBmkAscii^,INT_TO_STRING(BYTE_TO_INT(pstBMK^[iFor])-32));           // ASCII Nr - 32 wandelt klein- in Grossbuchstaben 
            iOfset                      := iOfset + 1;                                                                  // Zeichenversatz von + 1 je buchstaben 
        ELSIF BYTE_TO_INT(pstBMK^[iFor])= 45 THEN
            pstBmkAscii^[iFor + iOfset] := INT_TO_BYTE(43);     
        END_IF;
    END_FOR;
    //===========================================================================================================================================================================================================================================//
    //  Nr ergänzen 		                                                                          																															                 //
    //===========================================================================================================================================================================================================================================// 
    // Nr auf anzahl Stellen prüfen
    IF diNr >= 0 AND diNr <= 9 THEN
        IF xNoZero THEN
            stBmkAscii := CONCAT(stBMKAscii,DINT_TO_STRING(diNr));                                                      // Bei 1-Stelliger Zahl ohne 0 vorangesetzt
        ELSE
            stBmkAscii := CONCAT(stBMKAscii,CONCAT('0',DINT_TO_STRING(diNr)));                                          // Bei 1-Stelliger Zahl 0 voransetzen
        END_IF;    
    ELSIF diNr  >= 10 AND diNr <= 99 THEN
        stBmkAscii := CONCAT(stBMKAscii,DINT_TO_STRING(diNr));  
    ELSE
        IF enReportTypeIn = enReportType.Error THEN
            GVL_Report.fbReportVisu.proIdMissmatch := CONCAT(stBMK,CONCAT(' Error-ID not between 0-99 ID:',TO_STRING(diNr)));
        ELSIF enReportTypeIn = enReportType.Warning THEN
            GVL_Report.fbReportVisu.proIdMissmatch := CONCAT(stBMK,CONCAT(' Warning-ID not between 0-99 ID:',TO_STRING(diNr)));
        ELSIF enReportTypeIn = enReportType.Info THEN
            GVL_Report.fbReportVisu.proIdMissmatch := CONCAT(stBMK,CONCAT(' Info-ID not between 0-99 ID:',TO_STRING(diNr)));
        END_IF;    
    END_IF;
    //===========================================================================================================================================================================================================================================//
    //  Ausgabe DINT    		                                                                          																															             //
    //===========================================================================================================================================================================================================================================// 
    IF LEN(stBmkAscii) <= 12 THEN 
        fcBmkToId := TO_ULINT(stBMKAscii);
    ELSE 
        fcBmkToId := 0;
	END_IF
ELSE
    fcBmkToId   :=  TO_ULINT(diNr);    
END_IF;

END_FUNCTION

// 30 Program Organization Units/VIS/fbReportVisu
FUNCTION_BLOCK fbReportVisu 
VAR_INPUT
    ITF_BMK_IN                      :   ctaAppBmk.ITF_BMK;
END_VAR
VAR_OUTPUT
    xIsThereAnAktiveError           :   BOOL;
    xHandLokal                      :   BOOL;
END_VAR
VAR
    enVisuTableType                 :   enTableType;                                  
    ayItfReports                    :   ARRAY[0..GlobalKonstant.iUpperSizeTable] OF ITF_REPORTOBJECT;
    ayShowReport                    :   ARRAY[0..GlobalKonstant.iUpperSizeTable] OF BOOL;
    fbConfigFile                    :   CtaSysConfig.fbConfigFile;
    scPara                          :   scPara;
    ayReporter                      :   ARRAY[1..1] OF fbReporter;
    xFernQuitt                      :   BOOL;
    diFor                           :   DINT;
    iOffset                         :   INT;
    iOffsetOld                      :   INT;
    xReload                         :   BOOL;
	xWaitToReload					:	BOOL;
    xReloadExtern                   :   BOOL;
    xReloadIntern                   :   BOOL;
    iCountReadFromCsv               :   INT;
    xFirstLoadCsvDone               :   BOOL;  
    xFirstLoadPendingDone           :   BOOL; 
    udiMaxOffset                    :   UDINT;  
    xFilterError                    :   BOOL    := TRUE; 
    xFilterWarning                  :   BOOL    := TRUE;
    xFilterInfo                     :   BOOL    := TRUE;   
    usiFilter                       :   USINT;
    stIdMissmatch                   :   STRING;
END_VAR

actConfigFile();
(* Offset *)
IF iOffset <> iOffsetOld THEN
    xWaitToReload := TRUE;
ELSIF iOffset = iOffsetOld THEN
	IF xWaitToReload AND NOT xReloadExtern AND NOT xReloadIntern THEN
    	xReload 		:= TRUE;
		xWaitToReload 	:= FALSE;
	ELSE
		xReload 		:= FALSE;
		xWaitToReload 	:= FALSE;
	END_IF
END_IF;
iOffsetOld := iOffset;

IF enVisuTableType = enTableType.PENDING_REPORTS THEN
    (* Get Pending Reports *)
    actPending();   
    xFirstLoadCsvDone := FALSE;  
ELSIF enVisuTableType = enTableType.HISTORY_REPORTS THEN
    (* Get History CSV*)
    actHistory();    
    xFirstLoadPendingDone := FALSE;
    xFilterError          := TRUE;
    xFilterWarning        := TRUE;
    xFilterInfo           := TRUE;
END_IF;
  
actEWI();
xIsThereAnAktiveError := GVL_Report.fbReportObjectFactory.proIsThereAnAktiveError;
xHandLokal := GVL_Report.diCountHand <> 0;

METHOD metGetReport : ITF_REPORTOBJECT
VAR_INPUT
    iArrayPos   :   INT;
END_VAR
VAR
    xOk     :   BOOL;
END_VAR
metGetReport := 0;
IF iArrayPos >= 0 AND iArrayPos <= GlobalKonstant.iUpperSizeTable THEN
    IF __QUERYINTERFACE(ayItfReports[iArrayPos],metGetReport) THEN
        xOk := TRUE;    
    END_IF;
END_IF;
END_METHOD

METHOD metGetShowReport : BOOL
VAR_INPUT
    iArrayPos   :   INT;
END_VAR
IF iArrayPos >= 0 AND iArrayPos <= GlobalKonstant.iUpperSizeTable THEN
    metGetShowReport := ayShowReport[iArrayPos];
END_IF;
END_METHOD

ACTION actConfigFile:
(* PArameter *)
fbConfigFile();
scPara.fbxEnSafetyFernQuitt(_usiParaNr := 1,itfConfigFb:=fbConfigFile   ,_WertInit := TRUE);
scPara.fbuiMaxFernQuitt    (_usiParaNr := 2,itfConfigFb:=fbConfigFile   ,_WertInit := 5);
END_ACTION

PROPERTY proQuittExtern : BOOL
SET
IF proQuittExtern AND NOT xFernQuitt THEN
    IF scPara.fbxEnSafetyFernQuitt.proValue THEN
        IF ayReporter[1].proGetCounts < scPara.fbuiMaxFernQuitt.proValue THEN
            GVL_Report.fbReportObjectFactory.metQuittAllReports();
            xFernQuitt        := TRUE;
        END_IF;
    ELSE
        GVL_Report.fbReportObjectFactory.metQuittAllReports();
        xFernQuitt        := TRUE;
	END_IF;
ELSIF NOT proQuittExtern THEN
    xFernQuitt        := FALSE;
END_IF;
END_SET
END_PROPERTY

PROPERTY proMaxOffset : UDINT
GET
IF enVisuTableType = enTableType.PENDING_REPORTS THEN
    udiMaxOffset := LIMIT(0,TO_UDINT(proAnzReportsInTable),16#FFFFFFFF);
ELSIF enVisuTableType = enTableType.HISTORY_REPORTS THEN
    udiMaxOffset := GVL_Report.fbCsvHandler.proGetCountsOfReports;
END_IF
proMaxOffset := udiMaxOffset;
END_GET
END_PROPERTY

PROPERTY proOffset : INT
SET
iOffset     := proOffset;
END_SET
GET
proOffset := iOffset;
END_GET
END_PROPERTY

ACTION actEWI:
(* Externe Quittierung *)
ayReporter[1].metReport(xSetReportIn                := xFernQuitt,
                        iReportID                   := 99,
                        enReportTypeIn              := enReportType.Warning,
                        enReportAcknowledgeTypeIn   := SEL(scPara.fbxEnSafetyFernQuitt.proValue,enReportacknowledgeType.Auto,enReportacknowledgeType.RetryN),
                        tDelay                      := T#0S,
                        ITF_BMK_IN                  := ITF_BMK_IN,
                        pstReportTextListIn         := ADR(GlobalKonstant.stTextListWarning),
                        stOptionalReportText        := CONCAT(' ',TO_STRING(TO_INT(scPara.fbuiMaxFernQuitt.proValue)-(ayReporter[1].proGetCounts + 1))),
                        iRetryTilReportLock         := TO_INT(scPara.fbuiMaxFernQuitt.proValue),
                        xResetCount                 := FALSE,
                        tReset                      := T#1D);
END_ACTION

//FB_Init ist immer implizit verfügbar und wird primär für die Initialisierung verwendet.
//Der Rückgabewert wird nicht ausgewertet. Für gezielte Einflussnahme können Sie
//die Methoden explizit deklarieren und darin mit dem Standard-Initialisierungscode 
//zusätzlichen Code bereitstellen. Sie können den Rückgabewert auswerten.
METHOD FB_Init: BOOL
VAR_INPUT    
bInitRetains: BOOL; // TRUE: Die Retain-Variablen werden initialisiert (Reset warm / Reset kalt)    
bInCopyCode: BOOL;  // TRUE: Die Instanz wird danach in den Kopiercode kopiert (Online-Change)
END_VAR
END_METHOD

METHOD metReload : BOOL
VAR_INPUT
END_VAR
xReloadExtern := TRUE;
END_METHOD

ACTION actHistory:
(* Get ItF CSV*)
IF NOT xFirstLoadCsvDone OR xReload OR xReloadExtern THEN
    IF NOT xFirstLoadCsvDone THEN
        iOffset := 0;
	END_IF;
    FOR diFor := 0 TO GlobalKonstant.iUpperSizeTable DO
        IF __QUERYINTERFACE(GVL_Report.fbReportObjectFactory.metCsvGetItf(diFor),ayItfReports[diFor]) THEN
            ayItfReports[diFor].metDestroy();
            IF GVL_Report.fbCsvHandler.metReadCsv(ayItfReports[diFor],TO_DINT(promaxOffset - TO_UDINT(iOffset + diFor))) THEN   
                ayShowReport[diFor] := TRUE;   
            ELSE
                ayShowReport[diFor] := FALSE; 
            END_IF;      
        END_IF;
        IF diFor = GlobalKonstant.iUpperSizeTable THEN
            xFirstLoadCsvDone := TRUE;
        END_IF;
        xReloadExtern := FALSE;          
    END_FOR;
END_IF;
END_ACTION

ACTION actPending:
(* Get pending Reports *)
IF NOT xFirstLoadPendingDone OR xReload OR xReloadExtern OR xReloadIntern THEN
actCheckFilterAndSort();
GVL_Report.fbSort.metFilterCustom(usiFilter);
    IF NOT xFirstLoadPendingDone THEN
        iOffset := 0;
	END_IF;
    FOR diFor := 0 TO GlobalKonstant.iUpperSizeTable DO
        IF 1 + iOffset + diFor <= Parameter.diMaxObject THEN
            IF __QUERYINTERFACE(GVL_Report.ayItfSortetReportsCustom[1 + iOffset + diFor],ayItfReports[diFor]) THEN // Array Custom starts by 1 
                IF ayItfReports[diFor] <> 0 THEN   
                    ayShowReport[diFor] := TRUE;   
                ELSE
                    ayShowReport[diFor] := FALSE; 
                END_IF;      
            END_IF;
            IF diFor = GlobalKonstant.iUpperSizeTable THEN
                xFirstLoadPendingDone := TRUE;
            END_IF;
            xReloadIntern := FALSE;
            xReloadExtern := FALSE;     
        END_IF;     
    END_FOR;
END_IF;
END_ACTION

PROPERTY proFilterError : BOOL
GET
proFilterError := xFilterError;
END_GET
SET
xFilterError := proFilterError;
xReloadIntern := TRUE;
iOffset := 0;
END_SET
END_PROPERTY

PROPERTY proFilterWarning : BOOL
GET
proFilterWarning := xFilterWarning;
END_GET
SET
xFilterWarning := proFilterWarning;
xReloadIntern := TRUE;
iOffset := 0;
END_SET
END_PROPERTY

PROPERTY proFilterInfo : BOOL
GET
proFilterInfo := xFilterInfo;
END_GET
SET
xFilterInfo := proFilterInfo;
xReloadIntern := TRUE;
iOffset := 0;
END_SET
END_PROPERTY

ACTION actCheckFilterAndSort:
(* FILTER *) 
   (* No Filter *)
    IF xFilterError AND xFilterWarning AND xFilterInfo THEN
        usiFilter := 0;
    (* Only Error *)
    ELSIF xFilterError AND NOT xFilterWarning AND NOT xFilterInfo THEN
        usiFilter := 1;
    (* Only Warning *)    
    ELSIF NOT xFilterError AND xFilterWarning AND NOT xFilterInfo THEN
        usiFilter := 2;
    (* Only Info *)  
    ELSIF NOT xFilterError AND NOT xFilterWarning AND xFilterInfo THEN
        usiFilter := 3;    
    (* Error and Warning*)  
    ELSIF xFilterError AND xFilterWarning AND NOT xFilterInfo THEN
        usiFilter := 4;        
    (* Error and Info*)  
    ELSIF xFilterError AND NOT xFilterWarning AND xFilterInfo THEN
        usiFilter := 5;     
    (* Warning and Info*)  
    ELSIF NOT xFilterError AND xFilterWarning AND xFilterInfo THEN
        usiFilter := 6;   
    ELSE
        usiFilter := 0;
    END_IF;
END_ACTION

PROPERTY proAnzReportsInTable : UINT
GET
IF enVisuTableType = enTableType.PENDING_REPORTS THEN
    proAnzReportsInTable := GVL_Report.fbSort.proAnzReportsInTable;
ELSE
    proAnzReportsInTable := GVL_Report.fbSort.proAnzAktiveReports;
END_IF;
END_GET
END_PROPERTY

PROPERTY proIdMissmatch : STRING
SET
stIdMissmatch := proIdMissmatch;
END_SET
GET
proIdMissmatch := stIdMissmatch;
END_GET
END_PROPERTY

END_FUNCTION_BLOCK

// 30 Program Organization Units/SORT/fbSort
FUNCTION_BLOCK fbSort
VAR_INPUT
END_VAR
VAR_OUTPUT
END_VAR
VAR
    uiAnzAktivError             :   UINT;
    uiAnzAktivWarning           :   UINT;
    uiAnzAktivInfo              :   UINT;
    uiAnzAktivReports           :   UINT;
    uiAnzAktivReportsInTable    :   UINT;
END_VAR

METHOD metSortPrio : BOOL
VAR_INPUT
END_VAR
VAR
    diFor1    : DINT;
    diFor2    : DINT;
    itfTempt  : ITF_REPORTOBJECT;
    diCounts  : DINT;
END_VAR
(* Reset *)
FOR diFor1 := 1 TO Parameter.diMaxObject DO
		GVL_Report.ayItfAktiveReports[diFor1] := 0;
END_FOR;
uiAnzAktivError             := 0;
uiAnzAktivWarning           := 0;
uiAnzAktivInfo              := 0;
uiAnzAktivReports           := 0;

(* Get Aktive Reports *)
FOR diFor1 := 1 TO Parameter.diMaxObject DO
	IF GVL_Report.ayReportObject[diFor1].proStateActive THEN
		diCounts := LIMIT(1,diCounts + 1, Parameter.diMaxObject);
		GVL_Report.ayItfAktiveReports[diCounts] := GVL_Report.ayReportObject[diFor1];
		IF GVL_Report.ayItfAktiveReports[diCounts].proReportType = enReportType.Error THEN
			uiAnzAktivError     := uiAnzAktivError + 1;
		ELSIF GVL_Report.ayItfAktiveReports[diCounts].proReportType = enReportType.Warning THEN
			uiAnzAktivWarning   := uiAnzAktivWarning + 1;
		ELSIF GVL_Report.ayItfAktiveReports[diCounts].proReportType = enReportType.Info THEN
			uiAnzAktivInfo      := uiAnzAktivInfo + 1;
		END_IF
		uiAnzAktivReports := uiAnzAktivError + uiAnzAktivWarning + uiAnzAktivInfo;
	END_IF;
END_FOR;

(* Sort Aktive Reports dt *)
FOR diFor1 := 1 TO diCounts DO
	FOR diFor2 := 1 TO diCounts -1 DO
		(* Sort nach Typ *)
		IF GVL_Report.ayItfAktiveReports[diFor2].proDtFrom < GVL_Report.ayItfAktiveReports[diFor2 + 1].proDtFrom THEN
			itfTempt                                    := GVL_Report.ayItfAktiveReports[diFor2]; 
			GVL_Report.ayItfAktiveReports[diFor2]       := GVL_Report.ayItfAktiveReports[diFor2 + 1];
			GVL_Report.ayItfAktiveReports[diFor2 + 1]   := itfTempt;         
		END_IF;     
	END_FOR;
END_FOR

GVL_Report.ayItfSortetReportsPrio := GVL_Report.ayItfAktiveReports;
(* Sort *)
FOR diFor1 := 1 TO diCounts DO
	FOR diFor2 := 1 TO diCounts -1 DO
		(* Sort nach Typ *)
		IF __QUERYINTERFACE(GVL_Report.ayItfSortetReportsPrio[diFor2],GVL_Report.ayItfSortetReportsPrio[diFor2]) AND __QUERYINTERFACE(GVL_Report.ayItfSortetReportsPrio[diFor2 + 1],GVL_Report.ayItfSortetReportsPrio[diFor2 + 1]) THEN
			IF GVL_Report.ayItfSortetReportsPrio[diFor2].proReportType < GVL_Report.ayItfSortetReportsPrio[diFor2 + 1].proReportType THEN
				itfTempt                                        := GVL_Report.ayItfSortetReportsPrio[diFor2]; 
				GVL_Report.ayItfSortetReportsPrio[diFor2]       := GVL_Report.ayItfSortetReportsPrio[diFor2 + 1];
				GVL_Report.ayItfSortetReportsPrio[diFor2 + 1]   := itfTempt; 
			(* Sort nach Prio wenn Typ gleich *)    
			ELSIF GVL_Report.ayItfSortetReportsPrio[diFor2].proReportType = GVL_Report.ayItfSortetReportsPrio[diFor2 + 1].proReportType THEN
				IF GVL_Report.ayItfSortetReportsPrio[diFor2].proPrio > GVL_Report.ayItfSortetReportsPrio[diFor2 + 1].proPrio AND GVL_Report.ayItfSortetReportsPrio[diFor2 + 1].proPrio >= 1 THEN
					itfTempt                                        := GVL_Report.ayItfSortetReportsPrio[diFor2]; 
					GVL_Report.ayItfSortetReportsPrio[diFor2]       := GVL_Report.ayItfSortetReportsPrio[diFor2 + 1];
					GVL_Report.ayItfSortetReportsPrio[diFor2 + 1]   := itfTempt;                
				END_IF;           
			END_IF;     
		END_IF;
	END_FOR;
END_FOR;
GVL_Report.fbReportVisu.metReload();
END_METHOD

